// TwinCAT 3 PLC project tc_project_app
// ProgramVersion: 3.1.4026.16
// libraries:
//   Tc2_EtherCAT, * (Beckhoff Automation GmbH)
//   Tc2_MC2, * (Beckhoff Automation GmbH)
//   Tc2_NC, * (Beckhoff Automation GmbH)
//   Tc2_Standard, * (Beckhoff Automation GmbH)
//   Tc2_SUPS, * (Beckhoff Automation GmbH)
//   Tc2_System, * (Beckhoff Automation GmbH)
//   Tc2_Utilities, * (Beckhoff Automation GmbH)
//   Tc3_MC2_AdvancedHoming, * (Beckhoff Automation GmbH)
//   Tc3_Module, * (Beckhoff Automation GmbH)
//   VisuDialogs, * (System)
//   VisuSymbols,3.5.10.0,System
// project tree:
//   / GlobalTextList.TcGTLO (not stored), PlcTask.TcTTO (not stored), VisualizationManager.TcVMO (not stored)
//   GVLs/ GVL_APP.TcGVL, GVL_AxisNames.TcGVL
//   POUs/Application_Specific/Applications/ Application_Template.TcPOU (not stored), AxisTestProg.TcPOU
//   POUs/ MAIN.TcPOU
//   tc_mca_std_lib/DUTs/Axis_Structures/ ST_AxisConfig.TcDUT (not stored), ST_AxisControl.TcDUT (not stored), ST_AxisDescription.TcDUT (not stored), ST_AxisError.TcDUT (not stored), ST_AxisHomingConfig.TcDUT (not stored), ST_AxisInputs.TcDUT (not stored), ST_AxisPersistent.TcDUT (not stored), ST_AxisSPG.TcDUT (not stored), ST_AxisStatus.TcDUT (not stored), ST_AxisStruct.TcDUT (not stored)
//   tc_mca_std_lib/DUTs/ E_AxisParameters.TcTLEO (not stored), E_HomingRoutines.TcTLEO (not stored), E_AxisParameters.TcTLEO (not stored), E_RestorePosition.TcDUT (not stored), I_Axis.TcIO (not stored), E_SlitPairStatesV2.TcDUT (not stored), E_SlitPairStates.TcDUT (not stored), E_MotionFunctions.TcDUT (not stored), ST_McStatus.TcDUT (not stored)
//   tc_mca_std_lib/DUTs/Pneumatics/ E_PneumaticAxisErrors.TcDUT (not stored), E_PneumaticMode.TcDUT (not stored), ST_PneumaticAxisControl.TcDUT (not stored), ST_PneumaticAxisConfig.TcDUT (not stored), ST_PneumaticAxisInputs.TcDUT (not stored), ST_PneumaticAxisOutputs.TcDUT (not stored), ST_PneumaticAxisStatus.TcDUT (not stored), ST_PneumaticAxisStruct.TcDUT (not stored)
//   tc_mca_std_lib/GVLs/ GVL.TcGVL (not stored), GVL_UnitStrings.TcGVL (not stored)
//   tc_mca_std_lib/POUs/Motion/ FB_Axis.TcPOU, FB_SlitPair.TcPOU (not stored), FB_SlitPairV2.TcPOU (not stored), FB_SlitPairV3.TcPOU (not stored)
//   tc_mca_std_lib/POUs/Motion/Homing/ FB_Homing.TcPOU (not stored)
//   tc_mca_std_lib/POUs/Pneumatics/ FB_PneumaticAxis.TcPOU (not stored)
//   tc_mca_std_lib/Unused ESS Work/ E_AxisEngUnit.TcDUT (not stored), E_MonitoringLedFunction.TcDUT (not stored), FB_AxisTemperature.TcPOU (not stored), FB_ESSMonitoring.TcPOU (not stored), ST_MonitoringAlarm.TcDUT (not stored)
//   tc_mca_std_lib/VISUs/ MainVisu.TcVIS, ParameterTextList.TcTLO (not stored), PneumaticsVisu.TcVIS
// real-time tasks:
//   TASK PlcTask: cycle T#2ms, priority 10, ADS port 351
// motion (NC):
//   TASK NC-Task 1 SAF: cycle T#2ms, priority 4, ADS port 501
//   TASK NC-Task 1 SVB: cycle T#10ms, priority 8, ADS port 511
//   AXIS Axis 2 (id 2)
//     Dynamic: Acceleration=600, Deceleration=600
//     Velo: SlowManual=1, FastManual=3, Maximum=6
//     TargetPosControl: Range=0.005, Time=0.2
//     OtherSettings: AllowMotionCmdToSlave=true
//     encoder EncType=19
//       EncPara: ScaleFactorNumerator=5e-05, Offset=-351.3178, MaxCount=#xffffffff, ReferenceSystem=1
//         Inc: RefSoftSyncMask=#xffffffff
//     drive DrvType=24
//       Analog: VeloReferenz=6.25, VeloScale=0.95, TorqueSetpointScale=10, ScaleFactorActTorque=0.1
//       TimeComp: TaskDelayCycles=1
//     controller CtrType=1
//       CtrPara: PriorControlFactor=1
//         PosDiffControl: Range=1.5
//         PID: PosKp=4
//         Observer: BandWidth=20
// I/O:
//   DEVICE Device 1 (EtherCAT), AmsNetId 5.79.68.132.2.1
//     Term 1 (EK1200) [EK1200-5000 EtherCAT Power supply (2A E-Bus)]
//       Term 2 (EL1088) [EL1088 8Ch. Dig. Input 24V, 3ms, negative]
//       Term 3 (EL1808)
//       Term 4 (EL2819) [EL2819 16Ch. Dig. Output 24V, 0,5A, Diagnostic]
//       Term 5 (EK1110) [EK1110 EtherCAT extension]
//     Term 6 (EK1100) [EK1100 EtherCAT Coupler (2A E-Bus)]
//       Term 7 (EL3214) [EL3214 4Ch. Ana. Input PT100 (RTD)]
//       Term 8 (EL7047) [EL7047 1Ch. Stepper motor output stage (50V, 5A)]
//       Term 9 (EL7047) [EL7047 1Ch. Stepper motor output stage (50V, 5A)]
//       Term 10 (EL2008) [EL2008 8Ch. Dig. Output 24V, 0.5A]
//       Term 11 (EL7041-0052) [EL7041-0052 1Ch. Stepper motor output stage (50V, 5A)]
//       Term 12 (EL7041-1000) [EL7041-1000 1Ch. Stepper motor output stage (50V, 5A, standard)]
//       Term 13 (EL5042) [EL5042 2Ch. BiSS-C Encoder]
//       Term 28 (EL2008) [EL2008 8Ch. Dig. Output 24V, 0.5A]
//       Term 29 (EL1008) [EL1008 8Ch. Dig. Input 24V, 3ms]
//       Term 14 (EL9011) [EL9011 End Terminal]
// variable links:
//   (this object) <-> Device 1 (EtherCAT)/Term 6 (EK1100)/Term 13 (EL5042)
//     Enc/Inputs/In/nDataIn1 <-> FB Inputs Channel 1 compact/Position
//     Enc/Inputs/In/nState1 @bit 1 <-> FB Inputs Channel 1 compact/Status/Error
//     Enc/Inputs/In/nState1 @bit 2 <-> FB Inputs Channel 1 compact/Status/Ready
//     Enc/Inputs/In/nState1 <-> FB Inputs Channel 1 compact/Status/Warning
//     Enc/Inputs/In/nState2 @bit 4 <-> FB Inputs Channel 1 compact/Status/Diag
//     Enc/Inputs/In/nState2 @bit 6 <-> FB Inputs Channel 1 compact/Status/Input cycle counter
//     Enc/Inputs/In/nState2 @bit 5 <-> FB Inputs Channel 1 compact/Status/TxPDO State
//     Enc/Inputs/In/nState4 @bit 1 <-> WcState/InputToggle
//     Enc/Inputs/In/nState4 <-> WcState/WcState
//   (this object) <-> Device 1 (EtherCAT)/Term 6 (EK1100)/Term 9 (EL7047)
//     Drive/Inputs/In/nState1 @bit 3 <-> STM Status/Status/Error
//     Drive/Inputs/In/nState1 @bit 7 <-> STM Status/Status/Motor stall
//     Drive/Inputs/In/nState1 @bit 5 <-> STM Status/Status/Moving negative
//     Drive/Inputs/In/nState1 @bit 4 <-> STM Status/Status/Moving positive
//     Drive/Inputs/In/nState1 @bit 1 <-> STM Status/Status/Ready
//     Drive/Inputs/In/nState1 <-> STM Status/Status/Ready to enable
//     Drive/Inputs/In/nState1 @bit 6 <-> STM Status/Status/Torque reduced
//     Drive/Inputs/In/nState1 @bit 2 <-> STM Status/Status/Warning
//     Drive/Inputs/In/nState2 @bit 3 <-> STM Status/Status/Digital input 1
//     Drive/Inputs/In/nState2 @bit 4 <-> STM Status/Status/Digital input 2
//     Drive/Inputs/In/nState2 @bit 5 <-> STM Status/Status/Sync error
//     Drive/Inputs/In/nState2 @bit 7 <-> STM Status/Status/TxPDO Toggle
//     Drive/Inputs/In/nState4 @bit 1 <-> WcState/InputToggle
//     Drive/Inputs/In/nState4 <-> WcState/WcState
//     Drive/Outputs/Out/nCtrl1 <-> STM Control/Control/Enable
//     Drive/Outputs/Out/nCtrl1 @bit 2 <-> STM Control/Control/Reduce torque
//     Drive/Outputs/Out/nCtrl1 @bit 1 <-> STM Control/Control/Reset
//     Drive/Outputs/Out/nCtrl2 @bit 3 <-> STM Control/Control/Digital output 1
//     Drive/Outputs/Out/nDataOut2[0] <-> STM Velocity/Velocity
//   tc_project_app Instance <-> Device 1 (EtherCAT)/Term 6 (EK1100)/Term 28 (EL2008)
//     PlcTask Outputs/AxisTestProg.limitsPower <-> Channel 1/Output
//   tc_project_app Instance <-> Device 1 (EtherCAT)/Term 6 (EK1100)/Term 29 (EL1008)
//     PlcTask Inputs/GVL.astAxes[1].stInputs.bLimitBwd <-> Channel 2/Input
//     PlcTask Inputs/GVL.astAxes[1].stInputs.bLimitFwd <-> Channel 1/Input
//   tc_project_app Instance <-> NC-Task 1 SAF/Axes/Axis 2
//     PlcTask Inputs/GVL.astAxes[1].Axis.NcToPlc <-> Outputs/ToPlc
//     PlcTask Outputs/GVL.astAxes[1].Axis.PlcToNc <-> Inputs/FromPlc

// ---- GVLs/GVL_APP.TcGVL
{attribute 'qualified_only'}
VAR_GLOBAL
END_VAR

VAR_GLOBAL CONSTANT
    nAXIS_NUM: UINT := 8;
    nPNEUMATIC_AXIS_NUM: UINT := 0;
END_VAR

// ---- GVLs/GVL_AxisNames.TcGVL
VAR_GLOBAL
	MEASUREMENT_ANGLE : UINT := 1;
	HEIGHT_VIRTUAL : UINT:= 2;
	HEIGHT : UINT := 3;
	HORIZONTAL : UINT := 4;
	HORIZONTAL_VIRTUAL : UINT := 5;
	ROTATION_VIRTUAL : UINT := 6;
	ROTATION_LINEAR_REAL : UINT := 7;
	ROTATION_LINEAR_VIRTUAL_ENCODER : UINT := 8; //Encoder only axis to get speed information from
END_VAR

// ---- POUs/Application_Specific/Applications/AxisTestProg.TcPOU
PROGRAM AxisTestProg
VAR
    limitsPower AT %Q*: BOOL :=TRUE;
END_VAR

astAxes[1].stControl.bEnable:= TRUE;

END_PROGRAM

// ---- POUs/MAIN.TcPOU
PROGRAM MAIN
VAR
    sVersion: STRING := '1.0.0';
    aIAxes: ARRAY [1..GVL_APP.nAXIS_NUM] OF I_Axis;
    afbAxes: ARRAY [1..GVL_APP.nAXIS_NUM] OF FB_Axis;
    afbPneumaticAxes: ARRAY [1..GVL_APP.nPNEUMATIC_AXIS_NUM] OF FB_PneumaticAxis;
    hmiAxisSelection: INT := 1; //Not possible to use local hmi variables for array indexes
    hmiPneumaticAxisSelection: INT := 1;
//Startup, Shutdown and UPS
    fbUPS: FB_S_UPS_CX51x0;
    eUpsMode: E_S_UPS_Mode := eSUPS_WrPersistData_Shutdown;
    eStartUp: (eColdStart, eReadAxisFeedbackType, eCheckReadDone, eExecuteRestore, eCheckRestore, eFinishRestore);
    bPositionRestoreDone: BOOL := FALSE;
    bRestoreExecute: BOOL := FALSE;
	restoreCounter : UINT:=0;
	restoreCounterMax: UINT:=10;
    bExecuteReadEncRefSys: BOOL := FALSE;
    nRetry: INT;
    iAxes: UINT; //index for for loops in Position recovery actions
    afbReadEncRefSys: ARRAY [1..GVL_APP.nAXIS_NUM] OF MC_ReadParameter;
    afbSetPosition: ARRAY [1..GVL_APP.nAXIS_NUM] OF MC_SetPosition;
    afbReadPositionBias: ARRAY [1..GVL_APP.nAXIS_NUM] OF MC_ReadParameter;
    afbWritePositionBias: ARRAY [1..GVL_APP.nAXIS_NUM] OF MC_WriteParameter;
    fbGetDeviceIdentification: FB_GetDeviceIdentificationEx;
		
    tempAXOutput AT%Q* : BOOL:= TRUE;
	
	
END_VAR

VAR PERSISTENT
    bRestoreOnStartup: BOOL := TRUE;
END_VAR

//POSITION_RECOVERY();
RESTORE_POSITIONS();


IF bPositionRestoreDone THEN
	STORE_PERSISTENT();
END_IF


PROG();
AXES();

ACTION AXES:
//First cycle, assign FB_axis to interface array
IF _TaskInfo[fbGetCurTaskIndex.index].FirstCycle THEN
    FOR GVL.iAxis := 1 TO GVL_APP.nAXIS_NUM DO
        afbAxes[GVL.iAxis].stAxis REF= astAxes[GVL.iAxis];
        aIAxes[GVL.iAxis] := afbAxes[GVL.iAxis];
    END_FOR
    //Custom axis types defined and linked to aiAxes here
      //FB_CustomAxis extends FB_axis
        //fbCustomAxis.stAxis REF= astAxes[x];
        //aIAxes[x] := fbCustomAxis;
END_IF

//Execute FB_Axis logic
FOR GVL.iAxis := 1 TO GVL_APP.nAXIS_NUM DO
    aIAxes[GVL.iAxis].Run();
END_FOR

//Execute Pneumatic Axis logic
FOR GVL.iPneumaticAxis := 1 TO GVL_APP.nPNEUMATIC_AXIS_NUM DO
    afbPneumaticAxes[GVL.iPneumaticAxis](stPneumaticAxisStruct := GVL.astPneumaticAxes[GVL.iPneumaticAxis]);
END_FOR
END_ACTION

ACTION CHECK_UPS:
fbUPS(eUpsMode := eUpsMode);

FOR iAxes := 1 TO GVL_APP.nAXIS_NUM DO
    //Read encoder position BIAS
    IF astAxes[iAxes].stStatus.bAxisInitialized THEN
        afbReadPositionBias[iAxes](Axis := GVL.astAxes[iAxes].Axis,
                        Enable := TRUE,
                        ReadMode:= READMODE_CYCLIC,
                        ParameterNumber := E_AxisParameters.AxisEncoderOffset);
    END_IF
END_FOR

IF eGlobalSUpsState = eSUPS_PowerFailure THEN
    //first cycle of powerfailure
    //execute code that should only be done once with each powerfailure, i.e. increase powerfailure counter
    bRestoreOnStartup := TRUE;
    STORE_PERSISTENT();
    RETURN;
ELSIF eGlobalSUpsState <> eSUPS_PowerOK THEN
    //next cycles of powerfailure
    //skip regular code execution for the remaining cycles of the powerfailure/writing of persistent data/quick shutdown...
    RETURN;
END_IF
END_ACTION

ACTION POSITION_RECOVERY:
fbGetDeviceIdentification(bExecute := TRUE);
IF (fbGetDeviceIdentification.stDevIdent.strHardwareSerialNo <> '') THEN
    CHECK_UPS();
    RESTORE_POSITIONS();
END_IF
END_ACTION

ACTION PROG:
//Get task index for Axes parameters initialization.
GVL.fbGetCurTaskIndex();

//Call the programs that are defined in the "Application Specific" folder.
//Create as many programs in that folder as axes and applications you have or need

//Axes initial parameters and program
//Axis_Template();
//Pneumatics_Template();

//Application program calls
//Application_Template();
AxisTestProg();
END_ACTION

ACTION RESTORE_POSITIONS:
//This ACT will restore the position of an incremental axis on startup with the act position it read before losing power.
//It checks the type of axis, 0=incremental, and that the axis was stationary at shut down.
//Because 0 equates to incremental we also need to check that the data is valid, otherwise by default it would restore all axes.
//By default an axis will not restore the position unless it is set to opt-in, i.e. GVL.aAxes[iAxes].stConfig.eRestorePosition is non-zero.
//This needs to be initialised somewhere in TwinCAT code otherwise it will not be available at start up.
//A restore will only be performed on a loss of power, this code shouldn't make any changes on a reset cold, a rest origin or a download.
//There is a enum to allow for different types of restore modes, currently only one is implemented.
//0 'DontRestore'
//1 'RestoreWithoutHome' -restores the position using a set position fb and does not set the home bit in the axis struct.
//Note from Beckhoff: "A maximum of 1 MB persistent data can be reliably saved over the entire service life."
//Encoder Reference system types: https://infosys.beckhoff.com/english.php?content=../content/1033/tf50x0_tc3_nc_ptp/3439907723.html&id=
//INCREMENTAL=0;
//ABSOLUTE=1;
//ABSOLUTE (modulo)=2;
//ABSOLUTE MULTITURN RANGE (with single overflow)=3;
//INCREMENTAL (singleturn absolute)=4;
//ABSOLUTE SINGLETURN RANGE (with single overflow)=5;

IF NOT bPositionRestoreDone THEN
	bRestoreExecute := TRUE;
END_IF

//IF bRestoreOnStartup AND eGlobalSUpsState = eSUPS_PowerOK THEN
//    bRestoreOnStartup := FALSE;
//    bRestoreExecute := TRUE;
//END_IF

//Upon startup bPositionRestoreDone will be set to FALSE, after successfully completing the following code it will be set TRUE
//and should stay TRUE for the rest of the time the PLC is operational, thus this routine should only be completed once.
IF bRestoreExecute AND NOT bPositionRestoreDone THEN
    //Cycle through function blocks that read the encoder reference system i.e. whether axis is incremental or absolute
    FOR iAxes := 1 TO GVL_APP.nAXIS_NUM DO
         afbReadEncRefSys[iAxes](
            Axis := GVL.astAxes[iAxes].Axis,
            ParameterNumber := MC_AxisParameter.AxisEncoderReferenceSystem,
            ReadMode := E_READMODE.READMODE_ONCE);
    END_FOR

    //Cycle through set position and MC_WritePArameter function blocks for each axis
    FOR iAxes := 1 TO GVL_APP.nAXIS_NUM DO
        afbSetPosition[iAxes](
            Axis := GVL.astAxes[iAxes].Axis,
            Position := astAxesPersistent[iAxes].fPositionAtShutdown);

        afbWritePositionBias[iAxes](
            Axis:= GVL.astAxes[iAxes].Axis,
            ParameterNumber:= E_AxisParameters.AxisEncoderOffset,
            Value:= astAxesPersistent[iAxes].fEncoderBiasAtShutdown);
    END_FOR

    CASE eStartUp OF
        eColdStart:
            //First cycle of the PLC, do nothing just give one cycle for variables to initialise
            IF NOT bPositionRestoreDone THEN
                eStartUp := eReadAxisFeedbackType;
                nRetry := 0;
            END_IF

        eReadAxisFeedbackType:
            //Exectute the function blocks to read the encoder reference system (0=inc OR 1=ABS)
            FOR iAxes := 1 TO GVL_APP.nAXIS_NUM DO
                afbReadEncRefSys[iAxes].Enable := TRUE;
                eStartUp := eCheckReadDone;
            END_FOR

        eCheckReadDone:
            //Check the encoder reference system has been read for all axis -> if busy then continue with PLC cycle and check again next time.
            //If afbReadEncRefSys not started then go back a step.
            //If any axes result in an error the code will get stuck here, this happens if GVL_APP.nAXIS_NUM is not set correctly
            FOR iAxes := 1 TO GVL_APP.nAXIS_NUM DO
                IF NOT afbReadEncRefSys[iAxes].Valid THEN
                    IF afbReadEncRefSys[iAxes].Busy THEN
                        //Exit MAIN.STARTUP Action and wait till next cycle, needs to cycle through whole program in order for data to update
                        RETURN;
                    ELSE
                        //Sometimes the code gets here and the afbReadEncRefSys[iAxes] misses the rising edge. If  the code gets here it means
                        //valid=FALSE and .busy=FALSE which indicateds the FB probably hasn't started and thus needs to see a rising edge.
                        //Set execute to low, Exit MAIN.STARTUP and go back a step in the CASE statement.
                        afbReadEncRefSys[iAxes].Enable := FALSE;
                        eStartUp := eReadAxisFeedbackType;
                        nRetry := nRetry + 1; //counter used for troubleshooting to see how many cycles it takes before afbReadEncRefSys function blocks are read correctly
                        RETURN;
                    END_IF
                END_IF
            END_FOR
            //If the code gets here all axes have .valid=TRUE for all axes
            eStartUp := eExecuteRestore;

        eExecuteRestore:
            //Execute position and encoder BIAS restore by setting Execute = TRUE
           FOR iAxes := 1 TO GVL_APP.nAXIS_NUM DO
                IF GVL.astAxes[iAxes].stConfig.eRestorePosition = E_RestorePosition.eRestoreWithoutHome THEN
                    //Restore position value for incremental encoders
                    IF afbReadEncRefSys[iAxes].Value = 1 OR
                    afbReadEncRefSys[iAxes].Value = 3 OR
                    afbReadEncRefSys[iAxes].Value = 5 THEN
                       afbWritePositionBias[iAxes].Execute := TRUE;
					ELSIF NOT astAxesPersistent[iAxes].bMovingAtShutdown THEN
                       afbSetPosition[iAxes].Execute := TRUE;
                    //Restore encoder position BIAS for absolute encoders
                    
                    END_IF
                ELSE
                    RETURN;
                END_IF
            END_FOR
			restoreCounter:= restoreCounter+1;
            eStartUp := eCheckRestore;


        eCheckRestore:
            //Check the set position and write enocder BIAS fbs are finished
            //Nothing actually happens if the restore is not done, the code just returns from here each cycle and the
            //bPositionRestoreDone will never get set to TRUE and will take up cycle time
			IF restoreCounter>restoreCounterMax THEN
				eStartUp:= eFinishRestore;
				RETURN;
			END_IF
            eStartUp:= eFinishRestore;
			FOR iAxes := 1 TO GVL_APP.nAXIS_NUM DO
				
                IF GVL.astAxes[iAxes].stConfig.eRestorePosition = E_RestorePosition.eRestoreWithoutHome THEN
                    IF afbReadEncRefSys[iAxes].Value = 1 OR
                     afbReadEncRefSys[iAxes].Value = 3 OR
                     afbReadEncRefSys[iAxes].Value = 5 THEN
                        IF NOT afbWritePositionBias[iAxes].Done THEN
                            afbWritePositionBias[iAxes].Execute := FALSE;
                            eStartUp := eExecuteRestore;
                            RETURN;
                        END_IF
					ELSIF NOT astAxesPersistent[iAxes].bMovingAtShutdown THEN 
                        IF NOT afbSetPosition[iAxes].Done THEN
                            afbSetPosition[iAxes].Execute := FALSE;
                            eStartUp := eExecuteRestore;
                            RETURN;
                        END_IF
                     
                    END_IF
                END_IF
            END_FOR
            

        eFinishRestore:
            //Remove execute = TRUE for afbRestorePosition and fbWritePositionBias
            FOR iAxes := 1 TO GVL_APP.nAXIS_NUM DO
                afbSetPosition[iAxes].Execute := FALSE;
                afbWritePositionBias[iAxes].Execute := FALSE;
                bPositionRestoreDone := TRUE;
                bRestoreExecute := FALSE;
            END_FOR
    END_CASE
END_IF
END_ACTION

ACTION STORE_PERSISTENT:
FOR iAxes := 1 TO GVL_APP.nAXIS_NUM DO
    //Store Position beofre shutdown
    astAxesPersistent[iAxes].fPositionAtShutdown := GVL.astAxes[iAxes].Axis.NcToPlc.ActPos;

    //Store encoder position BIAS at shutdown
    astAxesPersistent[iAxes].fEncoderBiasAtShutdown := afbReadPositionBias[iAxes].Value;

    //Store value of moving at shutdown
    IF GVL.astAxes[iAxes].Axis.Status.StandStill OR GVL.astAxes[iAxes].Axis.Status.Disabled THEN
        astAxesPersistent[iAxes].bMovingAtShutdown := FALSE;
    ELSE
        astAxesPersistent[iAxes].bMovingAtShutdown := TRUE;
    END_IF
END_FOR
END_ACTION

END_PROGRAM

// ---- tc_mca_std_lib/POUs/Motion/FB_Axis.TcPOU
//Function block to run a virtual drive with Nc
FUNCTION_BLOCK FB_Axis IMPLEMENTS I_axis
VAR
    _stAxis: REFERENCE TO ST_AxisStruct; // Local property pointer for axis structure
    astMcStatus: ARRAY[1..nMCSTATUS_ARRAY_SIZE] OF POINTER TO ST_McStatus; //Array of all MC status signals defined in FB_init

    fbPower: MC_Power;
    stMcStatusPower: ST_McStatus;

    fbStop: MC_Stop;
    stMcStatusStop: ST_McStatus;

    fbHalt: MC_Halt;
    stMcStatusHalt: ST_McStatus;

    fbReset: MC_Reset;
    stMcStatusReset: ST_McStatus;

    fbMoveAbsolute: MC_MoveAbsolute;
    fbMoveAbsolute2: MC_MoveAbsolute;
    stMcStatusMoveAbsolute: ST_McStatus;

    fbMoveRelative: MC_MoveRelative;
    stMcStatusMoveRelative: ST_McStatus;

    fbMoveVelocity: MC_MoveVelocity;
    stMcStatusMoveVelocity: ST_McStatus;

    fbMoveModulo: MC_MoveModulo;
    fbMoveModulo2: MC_MoveModulo;
    stMcStatusMoveModulo: ST_McStatus;
	
	fbEnableSPG : MC_ExtSetPointGenEnable;
	stMcStatusEnableSPG : ST_McStatus;
	fbDisableSPG : MC_ExtSetPointGenDisable;
	stMcStatusDisableSPG : ST_McStatus;
	

    fbHome: FB_Homing;
    stMcStatusHome: ST_McStatus;

    fbReadParameter: MC_ReadParameter;
    stMcStatusReadParameter: ST_McStatus;

    fbWriteParameter: MC_WriteParameter;
    stMcStatusWriteParameter: ST_McStatus;
	
	fbSetPosition: MC_SetPosition;
	stMcStatusSetPosition: ST_McStatus;

    //Variables for holding limits during homing
    bWaitForStopAfterLimitHit: BOOL := FALSE;
    fbRemovePowerTimer: TOF;

    //Dedicated NC parameter read FBs
    fbReadAxisVeloManSlow: MC_ReadParameter;
    fbReadAxisVeloManFast: MC_ReadParameter;
    fbReadHomingVelToCam: MC_ReadParameter;
    fbReadHomingVelFromCam: MC_ReadParameter;
    fbReadAxisVeloMax: MC_ReadParameter;
    fbReadAxisMaxAcc: MC_ReadParameter;
    fbReadAxisMaxDec: MC_ReadParameter;
    fbReadAxisAcc: MC_ReadParameter;
    fbReadAxisDec: MC_ReadParameter;
    fbReadEnMinSoftPosLimit: MC_ReadParameter;
    fbReadEnMaxSoftPosLimit: MC_ReadParameter;
    fbReadMinSoftPosLimit: MC_ReadParameter;
    fbReadMaxSoftPosLimit: MC_ReadParameter;
    fbReadEnPositionLagMonitoring: MC_ReadParameter;
    fbReadAxisMaxPosLagValue: MC_ReadParameter;
    fbReadEnTargetPositionMonitoring: MC_ReadParameter;
    fbReadTargetPositionWindow: MC_ReadParameter;

    //Edge detection triggers for statuses
    fbDoneRTrig: R_TRIG;
    fbErrorRTrig: R_TRIG;
    fbCommandAbortedRTrig: R_TRIG;
    fbInVelocityRTrig: R_TRIG;
    fbInVelocityFTrig: F_TRIG;
    fbExecuteRTrig: R_TRIG;
    fbStopFinishedRiseEdge: R_TRIG;
    fbHaltFinishedRiseEdge: R_TRIG;
    fbResetFinishedRiseEdge: R_TRIG;
    fbAbsMovDyn1RiseEdge: R_TRIG;
    fbAbsMovDyn2RiseEdge: R_TRIG;
    fbModMovDyn1RiseEdge: R_TRIG;
    fbModMovDyn2RiseEdge: R_TRIG;
	
	fbMoveInProgressFTrig : F_TRIG;
	fbMoveInProgressEndTimer : TON;
	fbNewMoveRTrig : R_TRIG;
	bStartOfMove : BOOL;
	bEndOfMove : BOOL;
	
	bSpgEnableReq : BOOL;
	bSpgDisableReq : BOOL;
	spgDisableCommand : BOOL;

END_VAR
VAR CONSTANT
    nRATIO_DENOMINATOR_DEFAULT: UINT := 1;
    nNO_GEARING: UINT := 0;
    nMCSTATUS_ARRAY_SIZE: UINT := 12;
    nMULTI_MASTER_MAX_AXES: UINT := 4;
END_VAR

METHOD EndOfCycle : BOOL

_stAxis.stControl.bExecute := FALSE;
END_METHOD

METHOD FB_init : BOOL
VAR_INPUT
    bInitRetains: BOOL; // if TRUE, the retain variables are initialized (warm start / cold start)
    bInCopyCode: BOOL; // if TRUE, the instance afterwards gets moved into the copy code (online change)
END_VAR

//Copy address locations for statuses to an array to allow for easier checking of statuses
astMcStatus[1] := ADR(stMcStatusPower);
astMcStatus[2] := ADR(stMcStatusStop);
astMcStatus[3] := ADR(stMcStatusHalt);
astMcStatus[4] := ADR(stMcStatusReset);
astMcStatus[5] := ADR(stMcStatusMoveAbsolute);
astMcStatus[6] := ADR(stMcStatusMoveRelative);
astMcStatus[7] := ADR(stMcStatusMoveVelocity);
astMcStatus[8] := ADR(stMcStatusMoveModulo);
astMcStatus[9] := ADR(stMcStatusHome);
astMcStatus[10] := ADR(stMcStatusSetPosition);
astMcStatus[11] := ADR(stMcStatusReadParameter);
astMcStatus[12] := ADR(stMcStatusWriteParameter);
END_METHOD

METHOD mControl_AutoEnableDisable : BOOL
VAR_INPUT
END_VAR
//Has a move been requested?
IF _stAxis.stControl.eCommand = E_MotionFunctions.eMoveAbsolute OR 
	_stAxis.stControl.eCommand = E_MotionFunctions.eMoveModulo OR
	_stAxis.stControl.eCommand = E_MotionFunctions.eMoveRelative OR
	_stAxis.stControl.eCommand = E_MotionFunctions.eMoveVelocity OR
	_stAxis.stControl.eCommand = E_MotionFunctions.eHome THEN
	IF _stAxis.stControl.bExecute AND _stAxis.stStatus.bMoveRequested = FALSE THEN
		//new logic here to stop commands queuing with axes disabled if not meant to autoenable/disable
 		IF _stAxis.stStatus.bEnabled = FALSE AND _stAxis.stControl.bAutoEnableDisable = FALSE THEN
			_stAxis.stStatus.bMoveRequested := FALSE;
		ELSE
			_stAxis.stStatus.bMoveRequested := TRUE;
		END_IF
		//_stAxis.stStatus.bMoveRequested := TRUE;
	END_IF	
END_IF

IF _stAxis.stControl.bOverrideReadyToMove THEN
	_stAxis.stStatus.bReadyToMove := _stAxis.stControl.bExtReadyToMove;
ELSE
	_stAxis.stStatus.bReadyToMove := _stAxis.stStatus.bEnabled;
END_IF

IF fbMoveInProgressFTrig.Q THEN
	//start end move timer
	bEndOfMove:= TRUE;
	_stAxis.stControl.bExtReadyToMove:= FALSE;
END_IF
IF bStartOfMove THEN
	bEndOfMove:= FALSE;
	bStartOfMove:= FALSE;
END_IF

fbMoveInProgressEndTimer(IN:= bEndOfMove,PT:= _stAxis.stControl.tMoveFinishedDelay);

//If we want autoenabledisable
IF _stAxis.stControl.bAutoEnableDisable THEN
	//and a move has been requested and we are not enabled
	IF _stAxis.stStatus.bMoveRequested AND _stAxis.stStatus.bEnabled = FALSE THEN
		_stAxis.stControl.bEnable:= TRUE;
	END_IF
	IF _stAxis.stStatus.bMoveRequested = FALSE AND fbMoveInProgressEndTimer.Q THEN
	_stAxis.stControl.bEnable:= FALSE;
	bEndOfMove := FALSE;
	END_IF
END_IF

IF _stAxis.Axis.Status.Moving THEN
	_stAxis.stStatus.bMoveInProgress := TRUE;
END_IF

IF _stAxis.Axis.Status.NotMoving THEN
	_stAxis.stStatus.bMoveInProgress := FALSE;
END_IF

fbNewMoveRTrig(CLK:= _stAxis.stStatus.bMoveInProgress);
IF fbNewMoveRTrig.Q THEN
	bStartOfMove:= TRUE;
END_IF
fbMoveInProgressFTrig(CLK:= _stAxis.stStatus.bMoveInProgress OR spgDisableCommand);
//No move requested and no move in progress
END_METHOD

METHOD mControl_DisableSPG : BOOL
VAR_INPUT
END_VAR
IF _stAxis.stSpg.DisableSPG THEN
	//fbEnableSPG.Execute := TRUE;
	bSpgDisableReq := TRUE;
END_IF

IF _stAxis.stStatus.bEnabled = FALSE AND bSpgDisableReq THEN
	_stAxis.stStatus.messageString:= 'Axis is disabled';
	bSpgDisableReq:= FALSE;
END_IF

IF _stAxis.stStatus.SPGEnabled = FALSE AND bSpgDisableReq THEN
	stAxis.stStatus.messageString:= 'Axis is not in ExtSPG mode';
	bSpgDisableReq:= FALSE;
END_IF





fbDisableSPG.Execute:= bSpgDisableReq;
fbDisableSPG(Axis:= _stAxis.Axis);
IF _stAxis.stControl.bAutoEnableDisable THEN
	spgDisableCommand := fbDisableSPG.Done;
END_IF

_stAxis.stSpg.DisableSPG:= FALSE;
fbDisableSPG.Execute := FALSE;
END_METHOD

METHOD mControl_EnableSPG : BOOL
VAR_INPUT
END_VAR
IF _stAxis.stSpg.EnableSPG THEN
	//fbEnableSPG.Execute := TRUE;
	bSpgEnableReq := TRUE;
END_IF

IF _stAxis.stControl.bAutoEnableDisable = FALSE AND _stAxis.stStatus.bEnabled = FALSE AND bSpgEnableReq THEN
	_stAxis.stStatus.messageString:= 'Axis must be enabled before enabling ExtSPG';
	bSpgEnableReq:= FALSE;
END_IF

IF _stAxis.stControl.bAutoEnableDisable  AND _stAxis.stStatus.bEnabled = FALSE AND bSpgEnableReq = TRUE THEN
	_stAxis.stControl.bEnable:= TRUE;
END_IF


IF _stAxis.stStatus.bEnabled THEN
	fbEnableSPG.Execute := bSpgEnableReq;
	bSpgEnableReq := FALSE;
END_IF

fbEnableSPG(Axis:= _stAxis.Axis);

_stAxis.stSpg.EnableSPG:= FALSE;
fbEnableSPG.Execute := FALSE;
END_METHOD

METHOD mControl_FeedSPG : BOOL
VAR_INPUT
END_VAR

VAR
	DirectionInternal : DINT;
END_VAR
(* 
Direction 1 = Forward
Direction -1 = Backward
Direction 0 = Standstill
*)

IF _stAxis.stSpg.OverrideDirection THEN
	DirectionInternal:= _stAxis.stSpg.Direction;
ELSE
	//Direction calculation logic
	IF _stAxis.stSpg.Velocity > ABS(_stAxis.stSpg.VelocityStandstillThreshold) THEN
		DirectionInternal := 1;
	ELSIF _stAxis.stSpg.Velocity < -ABS(_stAxis.stSpg.VelocityStandstillThreshold) THEN
		DirectionInternal := -1;
	ELSE
		DirectionInternal := 0;
	END_IF
END_IF

MC_ExtSetPointGenFeed(
	Axis:= _stAxis.Axis, 
	Position:= _stAxis.stSpg.Position,
	Velocity:= _stAxis.stSpg.Velocity,
	Acceleration:= _stAxis.stSpg.Acceleration,
	Direction:= DirectionInternal);
END_METHOD

METHOD mControl_Home : ST_McStatus
IF _stAxis.stHomingConfig.eHomeSeq = E_HomingRoutines.eNoHoming THEN
    _stAxis.stStatus.bHomed := TRUE;
END_IF

IF _stAxis.stControl.eCommand = E_MotionFunctions.eHome THEN
    fbHome.bExecute := _stAxis.stControl.bExecute;
END_IF


fbHome.eHomeSeq := _stAxis.stHomingConfig.eHomeSeq;
fbHome.fHomePosition := _stAxis.stHomingConfig.fHomePosition;
fbHome.fHomeFinishDistance := _stAxis.stHomingConfig.fHomeFinishDistance;
fbHome(
    Axis := _stAxis.Axis,
    bLimitBwd := _stAxis.stInputs.bLimitBwd,
    bLimitFwd := _stAxis.stInputs.bLimitFwd,
    bHomeSensor := _stAxis.stInputs.bHomeSensor,
    stConfig := _stAxis.stConfig);
fbHome.bExecute := FALSE;

mControl_Home.Busy := fbHome.bBusy;
mControl_Home.CommandAborted := fbHome.bCommandAborted;
mControl_Home.Done := fbHome.bDone;
mControl_Home.Error := fbHome.bError;
mControl_Home.ErrorID := fbHome.nErrorId;

IF fbHome.bError THEN
    _stAxis.stError.nHomeErrorID := fbHome.nErrorID; //Set the error
END_IF
END_METHOD

METHOD mControl_LimitHitTimer : BOOL

//Timer for keeping power on after limit switch hit, needed for homing routines - if power is lost routines are aborted
fbRemovePowerTimer(IN := _stAxis.stInputs.bLimitFwd AND _stAxis.stInputs.bLimitBwd, PT := T#100MS);

IF stMcStatusHome.Busy AND (fbRemovePowerTimer.Q OR _stAxis.Axis.NcToPlc.AxisState = 5) THEN //5=PHASE_ACCNEG
    bWaitForStopAfterLimitHit := TRUE;
ELSE
    bWaitForStopAfterLimitHit := FALSE;
END_IF
END_METHOD

METHOD mControl_LimitLinking : BOOL

_stAxis.stStatus.bFwEnabled := _stAxis.stInputs.bLimitFwd OR _stAxis.stControl.bOverrideLimits; 
_stAxis.stStatus.bBwEnabled := _stAxis.stInputs.bLimitBwd OR _stAxis.stControl.bOverrideLimits;
_stAxis.stStatus.bInterlockedFwd := _stAxis.stControl.bInterlockFwd;
_stAxis.stStatus.bInterlockedBwd := _stAxis.stControl.bInterlockBwd;
END_METHOD

METHOD mControl_Power : ST_McStatus
fbPower.Enable := _stAxis.stControl.bEnable;

fbPower.Enable_Negative := (_stAxis.stStatus.bBwEnabled OR bWaitForStopAfterLimitHit) AND NOT _stAxis.stStatus.bInterlockedBwd;
fbPower.Enable_Positive := (_stAxis.stStatus.bFwEnabled OR bWaitForStopAfterLimitHit) AND NOT _stAxis.stStatus.bInterlockedFwd;
fbPower.Override := _stAxis.stConfig.fOverride;

fbPower(Axis := _stAxis.Axis);

mControl_Power.Error := fbPower.Error;

IF fbPower.Error THEN
    _stAxis.stError.nPowerErrorID := fbPower.ErrorID; //Set the error
END_IF
END_METHOD

METHOD mControl_Reset : ST_McStatus
VAR
    i: UINT;
END_VAR
fbReset.Execute := _stAxis.stControl.bReset;

fbReset(Axis := _stAxis.Axis);
IF fbReset.Done THEN
    _stAxis.stStatus.bError := FALSE;
	_stAxis.stStatus.bMcError := FALSE;
    FOR i := 1 TO nMCSTATUS_ARRAY_SIZE DO
        //Clear all the errors
        _stAxis.stStatus.nErrorID := 0;
    END_FOR
	_stAxis.stStatus.nMcErrorID := 0;
END_IF

mControl_Reset.Busy := fbReset.Busy;
mControl_Reset.Done := fbReset.Done;
mControl_Reset.Error := fbReset.Error;
mControl_Reset.ErrorID := fbReset.ErrorID;

IF fbReset.Error THEN
    _stAxis.stError.nResetErrorID := fbReset.ErrorID; //Set the error
END_IF

fbResetFinishedRiseEdge(CLK:=fbReset.Done OR fbReset.Error);
IF fbResetFinishedRiseEdge.Q OR fbReset.Done THEN
    _stAxis.stControl.bReset := FALSE;
END_IF
END_METHOD

METHOD mMove_Halt : ST_McStatus
fbHalt.Deceleration := _stAxis.stControl.fDeceleration;
fbHalt.Execute := _stAxis.stControl.bHalt;

fbHalt(Axis := _stAxis.Axis);

mMove_Halt.Busy := fbHalt.Busy;
mMove_Halt.Done := fbHalt.Done;
mMove_Halt.Error := fbHalt.Error;
mMove_Halt.ErrorID := fbHalt.ErrorID;
mMove_Halt.Active := fbHalt.Active;
mMove_Halt.CommandAborted := fbHalt.CommandAborted;

IF fbHalt.Error THEN
    _stAxis.stError.nHaltErrorID := fbHalt.ErrorID; //Set the error
END_IF

//Execution of fbHalt ended
fbHaltFinishedRiseEdge(CLK:=fbHalt.Done OR fbHalt.Error OR fbHalt.CommandAborted);
IF fbHaltFinishedRiseEdge.Q OR fbHalt.Done OR fbHalt.CommandAborted THEN
    _stAxis.stControl.bHalt := FALSE;
END_IF
END_METHOD

METHOD mMove_MoveAbsolute : ST_McStatus
IF _stAxis.stControl.eCommand = E_MotionFunctions.eMoveAbsolute THEN
	IF _stAxis.stStatus.bReadyToMove THEN
		fbMoveAbsolute.Execute := _stAxis.stStatus.bMoveRequested;
		IF _stAxis.stStatus.bMoveRequested THEN
			_stAxis.stStatus.bMoveRequested := FALSE;
		END_IF
    	IF fbMoveAbsolute.Execute AND fbMoveAbsolute.Busy THEN
        	fbMoveAbsolute2.Execute := TRUE;
    	END_IF
	END_IF    
END_IF

// Parameters
fbMoveAbsolute.Position := _stAxis.stControl.fPosition;
fbMoveAbsolute.Velocity := ABS(_stAxis.stControl.fVelocity);
fbMoveAbsolute.Acceleration := _stAxis.stControl.fAcceleration;
fbMoveAbsolute.Deceleration := _stAxis.stControl.fDeceleration;

fbMoveAbsolute2.Position := _stAxis.stControl.fPosition;
fbMoveAbsolute2.Velocity := ABS(_stAxis.stControl.fVelocity);
fbMoveAbsolute2.Acceleration := _stAxis.stControl.fAcceleration;
fbMoveAbsolute2.Deceleration := _stAxis.stControl.fDeceleration;


// Call both move absolute FB
fbMoveAbsolute(Axis := _stAxis.Axis);
fbMoveAbsolute2(Axis := _stAxis.Axis);

//Reset Execute bits
fbMoveAbsolute.Execute := FALSE;
fbMoveAbsolute2.Execute := FALSE;


// STATUS bits
mMove_MoveAbsolute.Active := fbMoveAbsolute.Active OR fbMoveAbsolute2.Active;
mMove_MoveAbsolute.Done := fbMoveAbsolute.Done OR fbMoveAbsolute2.Done;
mMove_MoveAbsolute.Busy := fbMoveAbsolute.Busy OR fbMoveAbsolute2.Busy;
mMove_MoveAbsolute.Error := fbMoveAbsolute.Error OR fbMoveAbsolute2.Error;


// Capture the CommandAborted for first scan if the other absolute move overtakes the current
fbAbsMovDyn1RiseEdge(CLK:= fbMoveAbsolute.Busy AND fbMoveAbsolute2.CommandAborted, Q=>);
fbAbsMovDyn2RiseEdge(CLK:= fbMoveAbsolute2.Busy AND fbMoveAbsolute.CommandAborted, Q=>);
mMove_MoveAbsolute.CommandAborted := (fbMoveAbsolute.CommandAborted AND NOT fbAbsMovDyn2RiseEdge.Q)
                                    OR (fbMoveAbsolute2.CommandAborted AND NOT fbAbsMovDyn1RiseEdge.Q);

// Error IDs
IF fbMoveAbsolute.Error THEN
    _stAxis.stError.nMoveAbsoluteErrorID := fbMoveAbsolute.ErrorID; //Set the error
    mMove_MoveAbsolute.ErrorID := fbMoveAbsolute.ErrorID;
END_IF
IF fbMoveAbsolute2.Error THEN
    _stAxis.stError.nMoveAbsoluteErrorID := fbMoveAbsolute2.ErrorID; //Set the error
    mMove_MoveAbsolute.ErrorID := fbMoveAbsolute2.ErrorID;
END_IF
END_METHOD

METHOD mMove_MoveModulo : ST_McStatus
IF _stAxis.stControl.eCommand = E_MotionFunctions.eMoveModulo THEN
	IF _stAxis.stStatus.bReadyToMove THEN
		fbMoveModulo.Execute := _stAxis.stStatus.bMoveRequested;
		IF _stAxis.stStatus.bMoveRequested THEN
			_stAxis.stStatus.bMoveRequested := FALSE;
		END_IF
    	IF fbMoveModulo.Execute AND fbMoveAbsolute.Busy THEN
        	fbMoveModulo2.Execute := TRUE;
    	END_IF
	END_IF    
END_IF

// Parameters
fbMoveModulo.Position := _stAxis.stControl.fPosition;
fbMoveModulo.Velocity := ABS(_stAxis.stControl.fVelocity);
fbMoveModulo.Acceleration := _stAxis.stControl.fAcceleration;
fbMoveModulo.Deceleration := _stAxis.stControl.fDeceleration;

fbMoveModulo2.Position := _stAxis.stControl.fPosition;
fbMoveModulo2.Velocity := ABS(_stAxis.stControl.fVelocity);
fbMoveModulo2.Acceleration := _stAxis.stControl.fAcceleration;
fbMoveModulo2.Deceleration := _stAxis.stControl.fDeceleration;

// Call both move absolute FB
fbMoveModulo(Axis := _stAxis.Axis);
fbMoveModulo.Execute := FALSE;
fbMoveModulo2(Axis := _stAxis.Axis);
fbMoveModulo2.Execute := FALSE;

// Status bits
mMove_MoveModulo.Active := fbMoveModulo.Active OR fbMoveModulo2.Active;
mMove_MoveModulo.Done := fbMoveModulo.Done OR fbMoveModulo2.Done;
mMove_MoveModulo.Busy := fbMoveModulo.Busy OR fbMoveModulo2.Busy;
mMove_MoveModulo.Error := fbMoveModulo.Error OR fbMoveModulo2.Error;

// Capture the CommandAborted for first scan if the other absolute move overtakes the current
fbModMovDyn1RiseEdge(CLK:= fbMoveModulo.Busy AND fbMoveModulo2.CommandAborted, Q=>);
fbModMovDyn2RiseEdge(CLK:= fbMoveModulo2.Busy AND fbMoveModulo.CommandAborted, Q=>);
mMove_MoveModulo.CommandAborted := (fbMoveModulo.CommandAborted AND NOT fbModMovDyn2RiseEdge.Q)
                                    OR (fbMoveModulo2.CommandAborted AND NOT fbModMovDyn1RiseEdge.Q);

// Error IDs
IF fbMoveModulo.Error THEN
    _stAxis.stError.nMoveModuloErrorID := fbMoveModulo.ErrorID; //Set the error
    mMove_MoveModulo.ErrorID := fbMoveModulo.ErrorID;
END_IF

IF fbMoveModulo2.Error THEN
    _stAxis.stError.nMoveModuloErrorID := fbMoveModulo2.ErrorID; //Set the error
    mMove_MoveModulo.ErrorID := fbMoveModulo2.ErrorID;
END_IF
END_METHOD

METHOD mMove_MoveRelative : ST_McStatus

IF _stAxis.stControl.eCommand = E_MotionFunctions.eMoveRelative THEN
	IF _stAxis.stStatus.bReadyToMove THEN
		fbMoveRelative.Execute := _stAxis.stStatus.bMoveRequested;
		IF _stAxis.stStatus.bMoveRequested THEN
			_stAxis.stStatus.bMoveRequested := FALSE;
		END_IF
	END_IF
END_IF

fbMoveRelative.Distance := _stAxis.stControl.fPosition;
fbMoveRelative.Velocity := ABS(_stAxis.stControl.fVelocity);
fbMoveRelative.Acceleration := _stAxis.stControl.fAcceleration;
fbMoveRelative.Deceleration := _stAxis.stControl.fDeceleration;

fbMoveRelative(Axis := _stAxis.Axis);
fbMoveRelative.Execute := FALSE;

mMove_MoveRelative.Active := fbMoveRelative.Active;
mMove_MoveRelative.Done := fbMoveRelative.Done;
mMove_MoveRelative.Busy := fbMoveRelative.Busy;
mMove_MoveRelative.Error := fbMoveRelative.Error;
mMove_MoveRelative.ErrorID := fbMoveRelative.ErrorID;
mMove_MoveRelative.CommandAborted := fbMoveRelative.CommandAborted;

IF fbMoveRelative.Error THEN
    _stAxis.stError.nMoveRelativeErrorID := fbMoveRelative.ErrorID; //Set the error
END_IF
END_METHOD

METHOD mMove_MoveVelocity : ST_McStatus

IF _stAxis.stControl.eCommand = E_MotionFunctions.eMoveVelocity THEN
	IF _stAxis.stStatus.bReadyToMove THEN
		fbMoveVelocity.Execute := _stAxis.stStatus.bMoveRequested;
		IF _stAxis.stStatus.bMoveRequested THEN
			_stAxis.stStatus.bMoveRequested := FALSE;
		END_IF
	END_IF
END_IF

fbMoveVelocity.Direction := SEL(_stAxis.stControl.fVelocity < 0, MC_Positive_Direction, MC_Negative_Direction);
fbMoveVelocity.Velocity := ABS(_stAxis.stControl.fVelocity);
fbMoveVelocity.Acceleration := _stAxis.stControl.fAcceleration;
fbMoveVelocity.Deceleration := _stAxis.stControl.fDeceleration;

fbMoveVelocity(Axis := _stAxis.Axis);
fbMoveVelocity.Execute:= FALSE;

mMove_MoveVelocity.Active := fbMoveVelocity.Active;
mMove_MoveVelocity.InVelocity := fbMoveVelocity.InVelocity;
mMove_MoveVelocity.Busy := fbMoveVelocity.Busy;
mMove_MoveVelocity.Error := fbMoveVelocity.Error;
mMove_MoveVelocity.ErrorID := fbMoveVelocity.ErrorID;
mMove_MoveVelocity.CommandAborted := fbMoveVelocity.CommandAborted;

IF fbMoveVelocity.Error THEN
    _stAxis.stError.nMoveVelocityErrorID := fbMoveVelocity.ErrorID; //Set the error
END_IF
END_METHOD

METHOD mMove_SetPosition : ST_McStatus
IF _stAxis.stControl.eCommand = E_MotionFunctions.eSetPosition THEN
	fbSetPosition.Execute:= _stAxis.stControl.bExecute;
END_IF

fbSetPosition.Position:= _stAxis.stControl.fPosition;
fbSetPosition.Options.ClearPositionLag:= TRUE;

fbSetPosition(Axis := _stAxis.Axis);
fbSetPosition.Execute:= FALSE;

mMove_SetPosition.Busy := fbSetPosition.Busy;
mMove_SetPosition.Error := fbSetPosition.Error;
mMove_SetPosition.ErrorID := fbSetPosition.ErrorID;
mMove_SetPosition.Done := fbSetPosition.Done;

IF fbSetPosition.Error THEN
    _stAxis.stError.nSetPositionErrorID := fbSetPosition.ErrorID; //Set the error
END_IF
END_METHOD

METHOD mMove_Stop : ST_McStatus
fbStop.Deceleration := _stAxis.stControl.fDeceleration;
fbStop.Execute := _stAxis.stControl.bStop;

fbStop(Axis := _stAxis.Axis);

mMove_Stop.Busy := fbStop.Busy;
mMove_Stop.Done := fbStop.Done;
mMove_Stop.Error := fbStop.Error;
mMove_Stop.ErrorID := fbStop.ErrorID;
mMove_Stop.Active := fbStop.Active;
mMove_Stop.CommandAborted := fbStop.CommandAborted;

IF fbStop.Error THEN
    _stAxis.stError.nStopErrorID := fbStop.ErrorID; //Set the error
END_IF

//Execution of fbStop ended
fbStopFinishedRiseEdge(CLK:=fbStop.Done OR fbStop.Error OR fbStop.CommandAborted);
IF fbStopFinishedRiseEdge.Q THEN
    _stAxis.stControl.bStop := FALSE;
END_IF
END_METHOD

METHOD mParameters_Init : BOOL
IF _stAxis.stControl.bReinitialiseNcParameters THEN
	_stAxis.stStatus.bAxisInitialized := FALSE;
	_stAxis.stControl.bReinitialiseNcParameters := FALSE;
END_IF
IF _stAxis.stConfig.bReadMcParametersValid AND NOT _stAxis.stStatus.bAxisInitialized THEN
    _stAxis.stControl.fAcceleration := _stAxis.stConfig.fDefaultAcc;
    _stAxis.stControl.fDeceleration := _stAxis.stConfig.fDefaultDec;
    _stAxis.stControl.fVelocity := _stAxis.stConfig.fVelocityDefaultFast;
    _stAxis.stControl.fJogVelocity := _stAxis.stConfig.fVelocityDefaultSlow;

    _stAxis.stStatus.bAxisInitialized := TRUE;
END_IF
END_METHOD

METHOD mParameters_ReadNc : BOOL

(*This act reads the MC parameters using an MC_ReadParameter FB FOR each variable
Intended TO be executed once every PLC cycle
Another FB is used TO trasnfer default axis parameters TO the stAxisStruct so
bReadValid is used TO halt that trasnfer UNTIL the parameters have been
read successfully. It may take a couple OF cycles once the PLC starts up.*)

//Slow jogging Velocity
fbReadAxisVeloManSlow(Axis := _stAxis.Axis,
                        Enable := TRUE,
                        ReadMode := READMODE_CYCLIC,
                        ParameterNumber := E_AxisParameters.AxisManualVelocitySlow,
                        Value => _stAxis.stConfig.fVelocityDefaultSlow);
//Fast jogging velocity
fbReadAxisVeloManFast(Axis := _stAxis.Axis,
                        Enable := TRUE,
                        ReadMode := READMODE_CYCLIC,
                        ParameterNumber := E_AxisParameters.AxisManualVelocityFast,
                        Value => _stAxis.stConfig.fVelocityDefaultFast);
//Homing velocity to Cam
fbReadHomingVelToCam(Axis := _stAxis.Axis,
                        Enable := TRUE,
                        ReadMode := READMODE_CYCLIC,
                        ParameterNumber := E_AxisParameters.AxisVelocityToCam,
                        Value => _stAxis.stHomingConfig.fHomingVelToCam);
//Homing velocity from Cam
fbReadHomingVelFromCam(Axis := _stAxis.Axis,
                        Enable := TRUE,
                        ReadMode := READMODE_CYCLIC,
                        ParameterNumber := E_AxisParameters.AxisVelocityFromCam,
                        Value => _stAxis.stHomingConfig.fHomingVelFromCam);
//Max velocity
fbReadAxisVeloMax(Axis := _stAxis.Axis,
                        Enable := TRUE,
                        ReadMode := READMODE_CYCLIC,
                        ParameterNumber := E_AxisParameters.AxisMaxVelocity,
                        Value => _stAxis.stConfig.fVeloMax);
//Max acceleration
fbReadAxisMaxAcc(Axis := _stAxis.Axis,
                        Enable := TRUE,
                        ReadMode := READMODE_CYCLIC,
                        ParameterNumber := E_AxisParameters.AxisMaximumAcceleration,
                        Value => _stAxis.stConfig.fMaxAcc);
//Max deceleration
fbReadAxisMaxDec(Axis := _stAxis.Axis,
                        Enable := TRUE,
                        ReadMode := READMODE_CYCLIC,
                        ParameterNumber := E_AxisParameters.AxisMaximumDeceleration,
                        Value => _stAxis.stConfig.fMaxDec);
//Default acceleration
fbReadAxisAcc(Axis := _stAxis.Axis,
                        Enable := TRUE,
                        ReadMode := READMODE_CYCLIC,
                        ParameterNumber := E_AxisParameters.AxisDefaultAcceleration,
                        Value => _stAxis.stConfig.fDefaultAcc);
//Default deceleration
fbReadAxisDec(Axis := _stAxis.Axis,
                        Enable := TRUE,
                        ReadMode := READMODE_CYCLIC,
                        ParameterNumber := E_AxisParameters.AxisDefaultDeceleration,
                        Value => _stAxis.stConfig.fDefaultDec);

//Soft limits enabled
fbReadEnMinSoftPosLimit(Axis := _stAxis.Axis,
                        Enable := TRUE,
                        ReadMode := READMODE_CYCLIC,
                        ParameterNumber := E_AxisParameters.EnableLimitBackward);
_stAxis.stConfig.bEnMinSoftPosLimit := LREAL_TO_BOOL(fbReadEnMinSoftPosLimit.Value);

fbReadEnMaxSoftPosLimit(Axis := _stAxis.Axis,
                        Enable := TRUE,
                        ReadMode := READMODE_CYCLIC,
                        ParameterNumber := E_AxisParameters.EnableLimitForward);
_stAxis.stConfig.bEnMaxSoftPosLimit := LREAL_TO_BOOL(fbReadEnMaxSoftPosLimit.Value);

//Soft limit values
fbReadMinSoftPosLimit(Axis := _stAxis.Axis,
                        Enable := TRUE,
                        ReadMode := READMODE_CYCLIC,
                        ParameterNumber := E_AxisParameters.SWLimitBackward,
                        Value => _stAxis.stConfig.fMinSoftPosLimit);
fbReadMaxSoftPosLimit(Axis := _stAxis.Axis,
                        Enable := TRUE,
                        ReadMode := READMODE_CYCLIC,
                        ParameterNumber := E_AxisParameters.SWLimitForward,
                        Value => _stAxis.stConfig.fMaxSoftPosLimit);

//Position Lag Monitoring
fbReadEnPositionLagMonitoring(Axis := _stAxis.Axis,
                        Enable := TRUE,
                        ReadMode := READMODE_CYCLIC,
                        ParameterNumber := E_AxisParameters.EnablePositionLagMonitoring);
_stAxis.stConfig.bEnPositionLagMonitoring := LREAL_TO_BOOL(fbReadEnPositionLagMonitoring.Value);

fbReadAxisMaxPosLagValue(Axis := _stAxis.Axis,
                        Enable := TRUE,
                        ReadMode := READMODE_CYCLIC,
                        ParameterNumber := E_AxisParameters.MaxPositionLag,
                        Value => _stAxis.stConfig.fMaxPosLagValue);

// Target Position Monitoring
fbReadEnTargetPositionMonitoring(Axis := _stAxis.Axis,
                        Enable := TRUE,
                        ReadMode := READMODE_CYCLIC,
                        ParameterNumber := E_AxisParameters.SWLimitBackward);
_stAxis.stConfig.bEnTargetPositionMonitoring := LREAL_TO_BOOL(fbReadEnTargetPositionMonitoring.Value);

fbReadTargetPositionWindow(Axis := _stAxis.Axis,
                        Enable := TRUE,
                        ReadMode := READMODE_CYCLIC,
                        ParameterNumber := E_AxisParameters.AxisTargetPositionWindow,
                        Value => _stAxis.stConfig.fTargetPositionWindow);

//All variables are valid
_stAxis.stConfig.bReadMcParametersValid := FALSE;
_stAxis.stConfig.bReadMcParametersValid := fbReadAxisVeloManSlow.Valid AND
    fbReadAxisVeloManFast.Valid AND
    fbReadHomingVelToCam.Valid AND
    fbReadHomingVelFromCam.Valid AND
    fbReadAxisVeloMax.Valid AND
    fbReadAxisAcc.Valid AND
    fbReadAxisDec.Valid AND
    fbReadEnMinSoftPosLimit.Valid AND
    fbReadEnMaxSoftPosLimit.Valid AND
    fbReadMinSoftPosLimit.Valid AND
    fbReadMaxSoftPosLimit.Valid AND
    fbReadEnPositionLagMonitoring.Valid AND
    fbReadAxisMaxPosLagValue.Valid AND
    fbReadEnTargetPositionMonitoring.Valid AND
    fbReadTargetPositionWindow.Valid;

//One of the variables has a read error
_stAxis.stConfig.bReadMcParametersError := fbReadAxisVeloManSlow.Error OR
    fbReadAxisVeloManFast.Error OR
    fbReadHomingVelToCam.Error OR
    fbReadHomingVelFromCam.Error OR
    fbReadAxisVeloMax.Error OR
    fbReadAxisAcc.Error OR
    fbReadAxisDec.Error OR
    fbReadEnMinSoftPosLimit.Error OR
    fbReadEnMaxSoftPosLimit.Error OR
    fbReadMinSoftPosLimit.Error OR
    fbReadMaxSoftPosLimit.Error OR
    fbReadEnPositionLagMonitoring.Error OR
    fbReadAxisMaxPosLagValue.Error OR
    fbReadEnTargetPositionMonitoring.Error OR
    fbReadTargetPositionWindow.Error;
END_METHOD

METHOD mParameters_ReadParameter : ST_McStatus

IF _stAxis.stControl.eCommand = E_MotionFunctions.eReadParameter THEN
    fbReadParameter.Enable := _stAxis.stControl.bExecute;
END_IF

fbReadParameter.ReadMode := E_READMODE.READMODE_ONCE;
fbReadParameter.ParameterNumber := _stAxis.stConfig.eAxisParameters;

fbReadParameter(Axis := _stAxis.Axis);
fbReadParameter.Enable := FALSE;

_stAxis.stconfig.fReadAxisParameter := fbReadParameter.Value;
mParameters_ReadParameter.Busy := fbReadParameter.Busy;
mParameters_ReadParameter.Done := fbReadParameter.Valid;
mParameters_ReadParameter.Error := fbReadParameter.Error;
mParameters_ReadParameter.ErrorID := fbReadParameter.ErrorID;

IF fbReadParameter.Error THEN
    _stAxis.stError.fbReadParameterErrorId := fbReadParameter.ErrorID;
END_IF
END_METHOD

METHOD mParameters_WriteParameter : ST_McStatus

IF _stAxis.stControl.eCommand = E_MotionFunctions.eWriteParameter THEN
    fbWriteParameter.Execute := _stAxis.stControl.bExecute;
END_IF

fbWriteParameter.ParameterNumber := _stAxis.stConfig.eAxisParameters;
fbWriteParameter.Value := _stAxis.stConfig.fWriteAxisParameter;

fbWriteParameter(Axis := _stAxis.Axis);
fbWriteParameter.Execute := FALSE;

mParameters_WriteParameter.Busy := fbWriteParameter.Busy;
mParameters_WriteParameter.Done := fbWriteParameter.Done;
mParameters_WriteParameter.Error := fbWriteParameter.Error;
mParameters_WriteParameter.ErrorID := fbWriteParameter.ErrorID;

IF fbWriteParameter.Error THEN
    _stAxis.stError.fbWriteParameterErrorId := fbWriteParameter.ErrorID;
END_IF
END_METHOD

METHOD mStatus_AxisStatus : BOOL

_stAxis.Axis.ReadStatus();
IF _stAxis.Axis.Status.OpMode.Modulo THEN
    _stAxis.stStatus.fActPosition := _stAxis.Axis.NcToPlc.ModuloActPos;
ELSE
    _stAxis.stStatus.fActPosition := _stAxis.Axis.NcToPlc.ActPos;
END_IF

_stAxis.stStatus.bHomed := _stAxis.Axis.Status.Homed;
_stAxis.stStatus.bMoving := _stAxis.Axis.Status.Moving;
_stAxis.stStatus.fActVelocity := _stAxis.Axis.NcToPlc.ActVelo;
_stAxis.stStatus.bMovingForward := _stAxis.Axis.Status.PositiveDirection;
_stAxis.stStatus.bMovingBackward := _stAxis.Axis.Status.NegativeDirection;
_stAxis.stStatus.bInTargetPosition := _stAxis.Axis.Status.InTargetPosition;
//_stAxis.stStatus.bEnabled := _stAxis.Axis.Status.Operational;
_stAxis.stStatus.bEnabled := NOT(_stAxis.Axis.Status.Disabled);	//This is crap but I don't know a better way

_stAxis.stStatus.SPGEnabled := _stAxis.Axis.Status.ExtSetPointGenEnabled;
END_METHOD

METHOD mStatus_Busy : BOOL
VAR
    i: UINT;
    tmpBusy: BOOL;
END_VAR

FOR i := 5 TO 10 DO
    tmpBusy := astMcStatus[i]^.Busy OR tmpBusy;
END_FOR
mStatus_Busy := tmpBusy;
END_METHOD

METHOD mStatus_CommandAborted : BOOL
VAR
    i: UINT;
    tmpCmdAborted: BOOL;
END_VAR

FOR i := 5 TO 9 DO
    tmpCmdAborted := astMcStatus[i]^.CommandAborted OR tmpCmdAborted;
END_FOR

fbCommandAbortedRTrig(CLK := tmpCmdAborted);
IF fbCommandAbortedRTrig.Q THEN
    _stAxis.stStatus.bCommandAborted := TRUE;
END_IF
END_METHOD

METHOD mStatus_Done : BOOL
VAR
    i: UINT;
    tmpDone: BOOL;
END_VAR

FOR i := 5 TO 10 DO
    tmpDone := astMcStatus[i]^.Done OR tmpDone;
END_FOR
//fbDoneRTrig(CLK:= mStatus_Done());
fbDoneRTrig(CLK := tmpDone);
IF fbDoneRTrig.Q THEN
    _stAxis.stStatus.bDone := TRUE;
END_IF
END_METHOD

METHOD mStatus_Error : BOOL
VAR
    i: UINT;
    tmpError: BOOL;
END_VAR

FOR i := 1 TO nMCSTATUS_ARRAY_SIZE DO
    tmpError := astMcStatus[i]^.Error OR tmpError;
END_FOR

fbErrorRTrig(CLK := tmpError);

//Check if NC is in error state and propogate
IF _stAxis.Axis.Status.ErrorStop OR _stAxis.Axis.Status.Error THEN
    _stAxis.stStatus.bError := _stAxis.Axis.Status.ErrorStop OR _stAxis.Axis.Status.Error;
    _stAxis.stStatus.nErrorID := _stAxis.Axis.Status.ErrorID;//NC Error ID
END_IF


IF fbErrorRTrig.Q THEN
        //For each mcStatus
        FOR i := 1 TO nMCSTATUS_ARRAY_SIZE DO
            //If there's an error present propagate
            IF astMcStatus[i]^.ErrorID <> 0 THEN
				_stAxis.stStatus.bMcError := TRUE;
                _stAxis.stStatus.nMcErrorID := astMcStatus[i]^.ErrorID;
            END_IF
        END_FOR
END_IF
END_METHOD

METHOD mStatus_InVelocity : BOOL
VAR
    i: UINT;
    tmpInVelocity: BOOL;
END_VAR
FOR i := 1 TO nMCSTATUS_ARRAY_SIZE DO
    tmpInVelocity := astMcStatus[i]^.InVelocity OR tmpInVelocity;
END_FOR
//fbInVelocityRTrig(CLK:= mStatus_InVelocity());
fbInVelocityRTrig(CLK := tmpInVelocity);
IF fbInVelocityRTrig.Q THEN
    _stAxis.stStatus.bInVelocity := TRUE;
END_IF

fbInVelocityFTrig(CLK := _stAxis.Axis.Status.ContinuousMotion);
IF fbInVelocityFTrig.Q THEN
    _stAxis.stStatus.bInVelocity := FALSE;
END_IF
END_METHOD

METHOD mStatus_NewCommand : BOOL
VAR
    i: UINT;
END_VAR

fbExecuteRTrig(CLK := _stAxis.stControl.bExecute);
IF fbExecuteRTrig.Q THEN
    _stAxis.stStatus.bDone := FALSE;
    _stAxis.stStatus.bCommandAborted := FALSE;

    //On a new motion command, clear the errorID
    CASE _stAxis.stControl.eCommand OF
            E_MotionFunctions.eMoveAbsolute,
            E_MotionFunctions.eMoveRelative,
            E_MotionFunctions.eMoveVelocity,
            E_MotionFunctions.eMoveModulo,
			E_MotionFunctions.eSetPosition,
            E_MotionFunctions.eHome :
                _stAxis.stStatus.nErrorID := 0;
            E_MotionFunctions.eWriteParameter,
            E_MotionFunctions.eReadParameter :
            // Nothing
    END_CASE
END_IF
END_METHOD

METHOD Run : BOOL
mStatus_AxisStatus();
mParameters_ReadNc();
mParameters_Init();
stMcStatusReadParameter := mParameters_ReadParameter();
stMcStatusWriteParameter := mParameters_WriteParameter();

mControl_LimitHitTimer();
mControl_LimitLinking();
stMcStatusPower := mControl_Power();
mControl_AutoEnableDisable();

mControl_EnableSPG();
mControl_DisableSPG();
mControl_FeedSPG();

stMcStatusHalt := mMove_Halt();
stMcStatusStop := mMove_Stop();
stMcStatusReset := mControl_Reset();
stMcStatusSetPosition := mMove_SetPosition();

stMcStatusMoveAbsolute := mMove_MoveAbsolute();
stMcStatusMoveRelative := mMove_MoveRelative();
stMcStatusMoveModulo := mMove_MoveModulo();
stMcStatusMoveVelocity := mMove_MoveVelocity();

stMcStatusHome := mControl_Home();

mStatus_NewCommand();
mStatus_Done();
mStatus_Error();
mStatus_InVelocity();
mStatus_CommandAborted();
_stAxis.stStatus.bBusy := mStatus_Busy();


EndOfCycle();
END_METHOD

PROPERTY stAxis : REFERENCE TO ST_AxisStruct
GET
stAxis REF= _stAxis;
END_GET
SET
_stAxis REF= stAxis;
END_SET
END_PROPERTY

END_FUNCTION_BLOCK

// ---- tc_mca_std_lib/VISUs/MainVisu.TcVIS
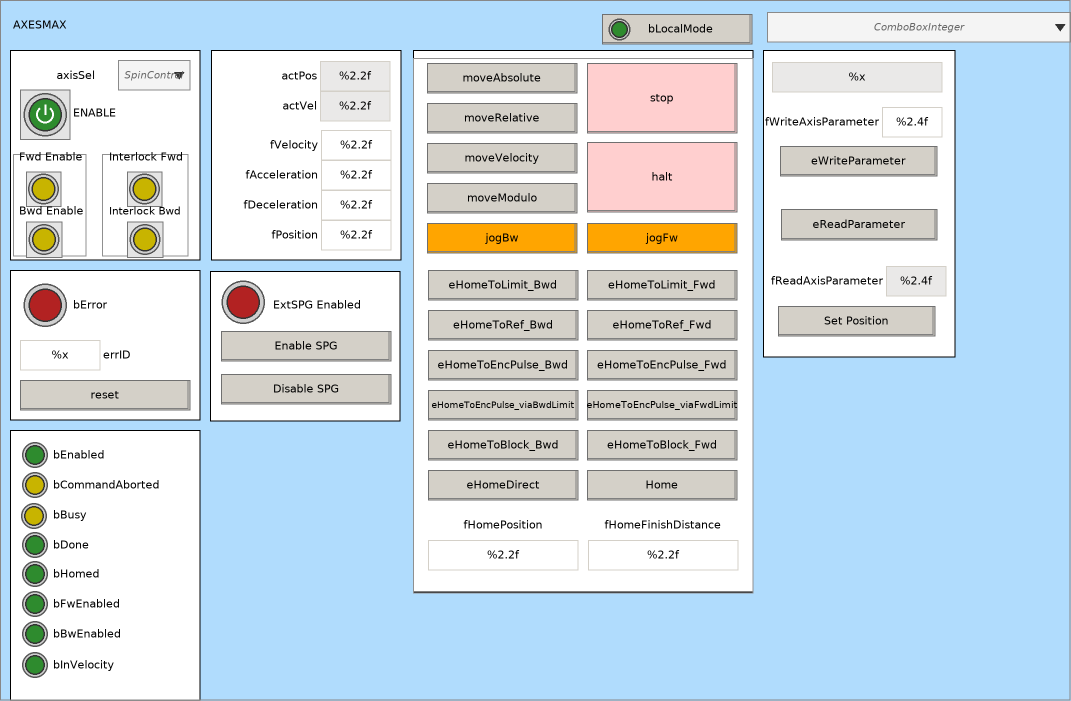
VISUALIZATION MainVisu  // 1071x701
    Rectangle (210,271 190x150)
    Rectangle (413,50 340x542)
    GroupBox (413,50 340x543)
        Button (174,92 150x70), "halt", pressed state: GVL.astAxes[Main.hmiAxisSelection].stControl.bHalt, text list: "languageSupport", text index: "halt"
            toggle GVL.astAxes[Main.hmiAxisSelection].stControl.bHalt
        Button (174,420 150x30), "Home", text list: 'languageSupport', text index: "Home"
            OnMouseClick: execute { GVL.astAxes[Main.hmiAxisSelection].stControl.eCommand:=E_MotionFunctions.eHome; GVL.astAxes[Main.hmiAxisSelection].stControl.bExecute:=TRUE; }
        Button (15,380 150x30), "eHomeToBlock_Bwd", text list: 'languageSupport', text index: "eHomeToBlock_Bwd"
            OnMouseClick: execute {
                GVL.astAxes[Main.hmiAxisSelection].stControl.eCommand:=E_MotionFunctions.eHome;
                GVL.astAxes[Main.hmiAxisSelection].stHomingConfig.eHomeSeq:=E_HomingRoutines.eHomeToBlock_Bwd;
                GVL.astAxes[Main.hmiAxisSelection].stControl.bExecute:=TRUE;
            }
    GroupBox (10,50 190x210)
        Rectangle (0,0 190x210)
        GroupBox (3,96 73x110)
        GroupBox (92,96 86x110)
        Textfield (60,50 92x26), "ENABLE", text list: 'languageSupport', text index: "enable"
        PushSwitchLed (16,118 35x42), variable: GVL.astAxes[MAIN.hmiAxisSelection].stInputs.bLimitFwd, behaviour: TOGGLE, style: Switch-PushSwitchLed-Yellow
        PushSwitchLed (16,170 36x39), variable: GVL.astAxes[MAIN.hmiAxisSelection].stInputs.bLimitBwd, behaviour: TOGGLE, style: Switch-PushSwitchLed-Yellow
        SpinControl (108,10 72x30), variable: MAIN.hmiAxisSelection
            p651134158: GVL_APP.nAXIS_NUM
        Textfield (23,13 86x25), "axisSel", text variable: GVL_APP.nAXIS_NUM, text list: "languageSupport", text index: "axisSel"
        PowerSwitch (10,38 50x53), variable: GVL.astAxes[MAIN.hmiAxisSelection].stControl.bEnable, behaviour: TOGGLE, style: Switch-PowerSwitch-Green
        PushSwitchLed (117,118 35x42), variable: GVL.astAxes[MAIN.hmiAxisSelection].stControl.bInterlockFwd, behaviour: TOGGLE, style: Switch-PushSwitchLed-Yellow
        PushSwitchLed (117,170 36x39), variable: GVL.astAxes[MAIN.hmiAxisSelection].stControl.bInterlockBwd, behaviour: TOGGLE, style: Switch-PushSwitchLed-Yellow
        Textfield (6,94 76x26), "Fwd Enable", text list: 'languageSupport', text index: "enFW"
        Textfield (6,148 76x26), "Bwd Enable", text list: 'languageSupport', text index: "enBW"
        Textfield (96,94 76x26), "Interlock Fwd", text list: 'languageSupport', text index: "bAxisInterlockFwd"
        Textfield (96,148 76x26), "Interlock Bwd", text list: 'languageSupport', text index: "bAxisInterlockBwd"
    Textfield (10,10 231x30), "AXESMAX", text variable: GVL_APP.nAXIS_NUM, text list: "languageSupport", text index: "axesAvailable"
    Button (427,63 150x30), "moveAbsolute", text list: "languageSupport", text index: "moveAbsolute"
        OnMouseClick: execute { GVL.astAxes[MAIN.hmiAxisSelection].stControl.eCommand:=E_MotionFunctions.eMoveAbsolute; GVL.astAxes[MAIN.hmiAxisSelection].stControl.bExecute:=TRUE; }
    Button (427,143 150x30), "moveVelocity", text list: "languageSupport", text index: "moveVelocity"
        OnMouseClick: execute { GVL.astAxes[Main.hmiAxisSelection].stControl.eCommand:=E_MotionFunctions.eMoveVelocity; GVL.astAxes[Main.hmiAxisSelection].stControl.bExecute:=TRUE; }
    Button (427,103 150x30), "moveRelative", text list: "languageSupport", text index: "moveRelative"
        OnMouseClick: execute { GVL.astAxes[Main.hmiAxisSelection].stControl.eCommand:=E_MotionFunctions.eMoveRelative; GVL.astAxes[Main.hmiAxisSelection].stControl.bExecute:=TRUE; }
    Button (427,183 150x30), "moveModulo", text list: "languageSupport", text index: "moveModulo"
        OnMouseClick: execute { GVL.astAxes[Main.hmiAxisSelection].stControl.eCommand:=E_MotionFunctions.eMoveModulo; GVL.astAxes[Main.hmiAxisSelection].stControl.bExecute:=TRUE; }
    Button (587,63 150x70), "stop", pressed state: GVL.astAxes[Main.hmiAxisSelection].stControl.bStop, text list: "languageSupport", text index: "stop"
        toggle GVL.astAxes[Main.hmiAxisSelection].stControl.bStop
    Button (427,223 150x30), "jogBw", text list: "languageSupport", text index: "jogBw"
        OnMouseDown: execute {
            GVL.astAxes[Main.hmiAxisSelection].stControl.eCommand:=E_MotionFunctions.eMoveVelocity;
            GVL.astAxes[Main.hmiAxisSelection].stControl.fVelocity:=-ABS(GVL.astAxes[Main.hmiAxisSelection].stControl.fJogVelocity)
            GVL.astAxes[Main.hmiAxisSelection].stControl.bExecute:= TRUE;
        }
        OnMouseClick: execute {  }
        OnMouseUp: execute { GVL.astAxes[Main.hmiAxisSelection].stControl.bHalt:= TRUE; }
    Button (587,223 150x30), "jogFw", text list: "languageSupport", text index: "jogFw"
        OnMouseDown: execute {
            GVL.astAxes[Main.hmiAxisSelection].stControl.eCommand:=E_MotionFunctions.eMoveVelocity;
            GVL.astAxes[Main.hmiAxisSelection].stControl.fVelocity:=ABS(GVL.astAxes[Main.hmiAxisSelection].stControl.fJogVelocity)
            GVL.astAxes[Main.hmiAxisSelection].stControl.bExecute:= TRUE;
        }
        OnMouseClick: execute {  }
        OnMouseUp: execute { GVL.astAxes[Main.hmiAxisSelection].stControl.bHalt:= TRUE; }
    GroupBox (10,270 190x150)
        Rectangle (0,0 190x150)
        Textfield (90,70 90x30), "errID", text list: "languageSupport", text index: "errID"
        Textfield (10,70 80x30), "%x", text variable: GVL.astAxes[MAIN.hmiAxisSelection].stStatus.nErrorID
        Lamp1 (10,10 50x50), variable: GVL.astAxes[MAIN.hmiAxisSelection].stStatus.bError, style: Lamp-Lamp1-Red
        Textfield (60,20 120x30), "bError", text list: "languageSupport", text index: "bError"
        Button (10,110 170x30), "reset", pressed state: GVL.astAxes[Main.hmiAxisSelection].stControl.bReset, text list: "languageSupport", text index: "reset"
            OnMouseClick: toggle GVL.astAxes[Main.hmiAxisSelection].stControl.bReset
    GroupBox (10,430 190x271)
        Rectangle (0,0 190x270)
        Lamp1 (10,10 30x30), variable: GVL.astAxes[MAIN.hmiAxisSelection].stStatus.bEnabled, style: Lamp-Lamp1-Green
        Textfield (40,10 140x30), "bEnabled", text list: "languageSupport", text index: "bEnabled"
        Lamp1 (10,40 30x30), variable: GVL.astAxes[MAIN.hmiAxisSelection].stStatus.bCommandAborted, style: Lamp-Lamp1-Yellow
        Textfield (40,40 140x30), "bCommandAborted", text list: "languageSupport", text index: "bWarning"
        Textfield (40,70 140x30), "bBusy", text list: "languageSupport", text index: "bBusy"
        Lamp1 (10,100 30x30), variable: GVL.astAxes[MAIN.hmiAxisSelection].stStatus.bDone, style: Lamp-Lamp1-Green
        Textfield (40,100 140x30), "bDone", text list: 'languageSupport', text index: "bDone"
        Lamp1 (10,129 30x30), variable: GVL.astAxes[MAIN.hmiAxisSelection].stStatus.bHomed, style: Lamp-Lamp1-Green
        Textfield (40,129 140x30), "bHomed", text list: "languageSupport", text index: "bHomed"
        Lamp1 (10,159 30x30), variable: GVL.astAxes[MAIN.hmiAxisSelection].stStatus.bFwEnabled AND NOT GVL.astAxes[MAIN.hmiAxisSelection].stStatus.bInterlockedFwd, style: Lamp-Lamp1-Green
        Lamp1 (10,189 30x30), variable: GVL.astAxes[MAIN.hmiAxisSelection].stStatus.bBwEnabled AND NOT GVL.astAxes[MAIN.hmiAxisSelection].stStatus.bInterlockedBwd, style: Lamp-Lamp1-Green
        Textfield (40,159 140x30), "bFwEnabled", text list: "languageSupport", text index: "bFwEnabled"
        Textfield (40,189 140x30), "bBwEnabled", text list: "languageSupport", text index: "bBwEnabled"
        Lamp1 (9,71 30x30), variable: GVL.astAxes[MAIN.hmiAxisSelection].stStatus.bBusy, style: Lamp-Lamp1-Yellow
        Lamp1 (10,220 30x30), variable: GVL.astAxes[MAIN.hmiAxisSelection].stStatus.bInVelocity, style: Lamp-Lamp1-Green
    GroupBox (211,50 190x210)
        Rectangle (0,0 190x210)
        Textfield (10,80 100x30), "fVelocity", text list: "languageSupport", text index: "fVelocity"
        Textfield (110,80 70x30), "%2.2f", text variable: GVL.astAxes[MAIN.hmiAxisSelection].stControl.fVelocity
            OnMouseClick: write the text variable via Default
        Textfield (10,110 100x30), "fAcceleration", text list: "languageSupport", text index: "fAcceleration"
        Textfield (110,110 70x30), "%2.2f", text variable: GVL.astAxes[MAIN.hmiAxisSelection].stControl.fAcceleration
            OnMouseClick: write the text variable via Default
        Textfield (10,140 100x30), "fDeceleration", text list: "languageSupport", text index: "fDeceleration"
        Textfield (110,140 70x30), "%2.2f", text variable: GVL.astAxes[MAIN.hmiAxisSelection].stControl.fDeceleration
            OnMouseClick: write the text variable via Default
        Textfield (10,170 100x30), "fPosition", text list: "languageSupport", text index: "fPosition"
        Textfield (110,170 70x30), "%2.2f", text variable: GVL.astAxes[MAIN.hmiAxisSelection].stControl.fPosition
            OnMouseClick: write the text variable via Default
        Textfield (109,11 70x30), "%2.2f", text variable: GVL.astAxes[MAIN.hmiAxisSelection].stStatus.fActPosition
        Textfield (9,11 100x30), "actPos", text list: "languageSupport", text index: "actposition"
        Textfield (9,41 100x30), "actVel", text list: "languageSupport", text index: "actVelocity"
        Textfield (109,41 70x30), "%2.2f", text variable: GVL.astAxes[MAIN.hmiAxisSelection].stStatus.fActVelocity
    Button (428,310 150x30), "eHomeToRef_Bwd", text list: 'languageSupport', text index: "eHomeToRef_Bwd"
        OnMouseClick: execute {
            GVL.astAxes[Main.hmiAxisSelection].stControl.eCommand:=E_MotionFunctions.eHome;
            GVL.astAxes[Main.hmiAxisSelection].stHomingConfig.eHomeSeq:=E_HomingRoutines.eHomeToRef_Bwd;
            GVL.astAxes[Main.hmiAxisSelection].stControl.bExecute:=TRUE;
        }
    Button (587,310 150x30), "eHomeToRef_Fwd", text list: "languageSupport", text index: "eHomeToRef_Fwd"
        OnMouseClick: execute {
            GVL.astAxes[Main.hmiAxisSelection].stControl.eCommand:=E_MotionFunctions.eHome;
            GVL.astAxes[Main.hmiAxisSelection].stHomingConfig.eHomeSeq:=E_HomingRoutines.eHomeToRef_Fwd;
            GVL.astAxes[Main.hmiAxisSelection].stControl.bExecute:=TRUE;
        }
    Button (428,350 150x30), "eHomeToEncPulse_Bwd", text list: 'languageSupport', text index: "eHomeToEncPulse_Bwd"
        OnMouseClick: execute {
            GVL.astAxes[Main.hmiAxisSelection].stControl.eCommand:=E_MotionFunctions.eHome;
            GVL.astAxes[Main.hmiAxisSelection].stHomingConfig.eHomeSeq:=E_HomingRoutines.eHomeToEncPulse_Bwd;
            GVL.astAxes[Main.hmiAxisSelection].stControl.bExecute:=TRUE;
        }
    Button (587,350 150x30), "eHomeToEncPulse_Fwd", text list: "languageSupport", text index: "eHomeToEncPulse_Fwd"
        OnMouseClick: execute {
            GVL.astAxes[Main.hmiAxisSelection].stControl.eCommand:=E_MotionFunctions.eHome;
            GVL.astAxes[Main.hmiAxisSelection].stHomingConfig.eHomeSeq:=E_HomingRoutines.eHomeToEncPulse_Fwd;
            GVL.astAxes[Main.hmiAxisSelection].stControl.bExecute:=TRUE;
        }
    Button (428,470 150x30), "eHomeDirect", text list: 'languageSupport', text index: "eHomeDirect"
        OnMouseClick: execute {
            GVL.astAxes[Main.hmiAxisSelection].stControl.eCommand:=E_MotionFunctions.eHome;
            GVL.astAxes[Main.hmiAxisSelection].stHomingConfig.eHomeSeq:=E_HomingRoutines.eHomeDirect;
            GVL.astAxes[Main.hmiAxisSelection].stControl.bExecute:=TRUE;
        }
    Button (428,270 150x30), "eHomeToLimit_Bwd", text list: 'languageSupport', text index: "eHomeToLimit_Bwd"
        OnMouseClick: execute {
            GVL.astAxes[Main.hmiAxisSelection].stControl.eCommand:=E_MotionFunctions.eHome;
            GVL.astAxes[Main.hmiAxisSelection].stHomingConfig.eHomeSeq:=E_HomingRoutines.eHomeToLimit_Bwd;
            GVL.astAxes[Main.hmiAxisSelection].stControl.bExecute:=TRUE;
        }
    Button (587,270 150x30), "eHomeToLimit_Fwd", text list: "languageSupport", text index: "eHomeToLimit_Fwd"
        OnMouseClick: execute {
            GVL.astAxes[Main.hmiAxisSelection].stControl.eCommand:=E_MotionFunctions.eHome;
            GVL.astAxes[Main.hmiAxisSelection].stHomingConfig.eHomeSeq:=E_HomingRoutines.eHomeToLimit_Fwd;
            GVL.astAxes[Main.hmiAxisSelection].stControl.bExecute:=TRUE;
        }
    Textfield (428,540 150x30), "%2.2f", text variable: GVL.astAxes[MAIN.hmiAxisSelection].stHomingConfig.fHomePosition
        OnMouseClick: write GVL.astAxes[MAIN.hmiAxisSelection].stHomingConfig.fHomePosition via Default
    Button (428,390 150x30), "eHomeToEncPulse_viaBwdLimit", text list: 'languageSupport', text index: "eHomeToEncPulse_viaBwdLimit"
        OnMouseClick: execute {
            GVL.astAxes[Main.hmiAxisSelection].stControl.eCommand:=E_MotionFunctions.eHome;
            GVL.astAxes[Main.hmiAxisSelection].stHomingConfig.eHomeSeq:=E_HomingRoutines.eHomeToEncPulse_viaBwdLimit;
            GVL.astAxes[Main.hmiAxisSelection].stControl.bExecute:=TRUE;
        }
    Button (587,390 150x30), "eHomeToEncPulse_viaFwdLimit", text list: "languageSupport", text index: "eHomeToEncPulse_viaFwdLimit"
        OnMouseClick: execute {
            GVL.astAxes[Main.hmiAxisSelection].stControl.eCommand:=E_MotionFunctions.eHome;
            GVL.astAxes[Main.hmiAxisSelection].stHomingConfig.eHomeSeq:=E_HomingRoutines.eHomeToEncPulse_viaFwdLimit;
            GVL.astAxes[Main.hmiAxisSelection].stControl.bExecute:=TRUE;
        }
    Textfield (588,540 150x30), "%2.2f", text variable: GVL.astAxes[MAIN.hmiAxisSelection].stHomingConfig.fHomeFinishDistance, text list: ''
        OnMouseClick: write GVL.astAxes[MAIN.hmiAxisSelection].stHomingConfig.fHomeFinishDistance via Default
    Textfield (428,510 150x30), "fHomePosition", text list: "languageSupport", text index: "fHomePosition"
    Textfield (588,510 150x30), "fHomeFinishDistance", text list: "languageSupport", text index: "fHomeFinishDistance"
    Group (602,14 150x30)
        Button (0,0 150x30), "bLocalMode", text list: 'languageSupport', text index: bLocalMode
            OnMouseClick: toggle bLocalMode
        Lamp1 (5,3 25x25), variable: bLocalMode, style: Lamp-Lamp1-Green
    Rectangle (763,50 192x307)
    Button (780,146 157x30), "eWriteParameter", text list: "languageSupport", text index: "eWriteParameter"
        OnMouseClick: execute { GVL.astAxes[MAIN.hmiAxisSelection].stControl.eCommand:=E_MotionFunctions.eWriteParameter; GVL.astAxes[MAIN.hmiAxisSelection].stControl.bExecute:=TRUE; }
    Textfield (772,62 170x30), "%x", text variable: astAxes[MAIN.hmiAxisSelection].stConfig.eAxisParameters
        OnMouseClick: write GVL.astAxes[MAIN.hmiAxisSelection].stConfig.eAxisParameters via Default
    Textfield (762,107 120x30), "fWriteAxisParameter", text list: "languageSupport", text index: "fWriteAxisParameter"
    Textfield (882,107 60x30), "%2.4f", text variable: astAxes[MAIN.hmiAxisSelection].stConfig.fWriteAxisParameter
        OnMouseClick: write GVL.astAxes[MAIN.hmiAxisSelection].stConfig.fWriteAxisParameter via Default
    Textfield (886,266 60x30), "%2.4f", text variable: astAxes[MAIN.hmiAxisSelection].stConfig.fReadAxisParameter
        OnMouseClick: write GVL.astAxes[MAIN.hmiAxisSelection].stConfig.fReadAxisParameter via Default
    Textfield (766,266 120x30), "fReadAxisParameter", text list: "languageSupport", text index: "fReadAxisParameter"
    Button (781,209 156x31), "eReadParameter", text list: 'languageSupport', text index: "eReadParameter"
        OnMouseClick: execute { GVL.astAxes[MAIN.hmiAxisSelection].stControl.eCommand:=E_MotionFunctions.eReadParameter; GVL.astAxes[MAIN.hmiAxisSelection].stControl.bExecute:=TRUE; }
    ComboBoxInteger (767,12 304x30), variable: GVL.astAxes[MAIN.hmiAxisSelection].stConfig.eAxisParameters, text list: 'ParameterTextList'
    Textfield (50,650 140x30), "bInVelocity", text list: 'languageSupport', text index: "bInVelocity"
    Button (587,430 150x30), "eHomeToBlock_Fwd", text list: "languageSupport", text index: "eHomeToBlock_Fwd"
        OnMouseClick: execute {
            GVL.astAxes[Main.hmiAxisSelection].stControl.eCommand:=E_MotionFunctions.eHome;
            GVL.astAxes[Main.hmiAxisSelection].stHomingConfig.eHomeSeq:=E_HomingRoutines.eHomeToBlock_Fwd;
            GVL.astAxes[Main.hmiAxisSelection].stControl.bExecute:=TRUE;
        }
    Textfield (270,290 120x30), "ExtSPG Enabled", text list: "languageSupport", text index: "bError"
    Lamp1 (218,277 50x50), variable: GVL.astAxes[MAIN.hmiAxisSelection].stStatus.SPGEnabled, style: Lamp-Lamp1-Red
    Button (221,331 170x30), "Enable SPG", pressed state: GVL.astAxes[Main.hmiAxisSelection].stControl.bReset, text list: "languageSupport", text index: "reset"
        OnMouseClick: toggle GVL.astAxes[Main.hmiAxisSelection].stSpg.EnableSPG
    Button (221,374 170x30), "Disable SPG", pressed state: GVL.astAxes[Main.hmiAxisSelection].stControl.bReset, text list: "languageSupport", text index: "reset"
        OnMouseClick: toggle GVL.astAxes[Main.hmiAxisSelection].stSpg.DisableSPG
    Button (778,306 157x30), "Set Position", text list: "languageSupport", text index: "eWriteParameter"
        OnMouseClick: execute { GVL.astAxes[MAIN.hmiAxisSelection].stControl.eCommand:=E_MotionFunctions.eSetPosition; GVL.astAxes[MAIN.hmiAxisSelection].stControl.bExecute:=TRUE; }
END_VISUALIZATION

// ---- tc_mca_std_lib/VISUs/PneumaticsVisu.TcVIS
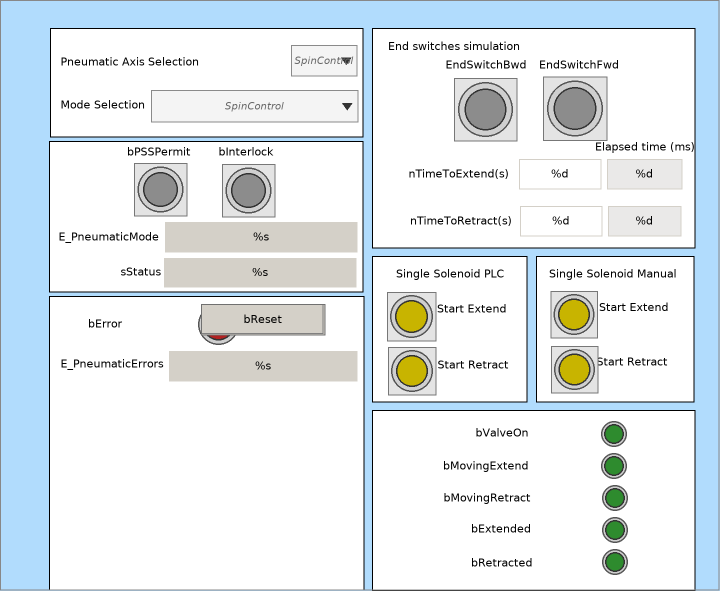
VISUALIZATION PneumaticsVisu  // 720x591
    Rectangle (50,28 313x109)
    Label (55,47 150x30), "Pneumatic Axis Selection"
    Rectangle (372,28 323x220)
    Label (379,30 150x33), "End switches simulation"
    Label (411,50 150x30), "EndSwitchBwd"
    SpinControl (291,45 66x31), variable: MAIN.hmiPneumaticAxisSelection
        p651134158: GVL_APP.nPNEUMATIC_AXIS_NUM
    Label (504,50 150x30), "EndSwitchFwd"
    Rectangle (49,296 315x294)
    Textfield (519,159 82x30), "%d", text variable: MAIN.afbPneumaticAxes[MAIN.hmiPneumaticAxisSelection].stPneumaticAxisStruct.stPneumaticAxisConfig.nTimeToExtend
        OnMouseClick: write MAIN.afbPneumaticAxes[MAIN.hmiPneumaticAxisSelection].stPneumaticAxisStruct.stPneumaticAxisConfig.nTimeToExtend via Default
    Label (384,159 150x30), "nTimeToExtend(s)"
    Label (386,206 150x30), "nTimeToRetract(s)"
    Label (28,90 150x30), "Mode Selection"
    Rectangle (49,141 314x151)
    Label (30,309 150x30), "bError"
    Lamp1 (126,301 185x47), variable: MAIN.afbPneumaticAxes[MAIN.hmiPneumaticAxisSelection].stPneumaticAxisStruct.stPneumaticAxisStatus.bError, style: Lamp-Lamp1-Red
    Label (37,349 150x30), "E_PneumaticErrors"
    Textfield (169,351 188x30), "%s", text variable: MAIN.afbPneumaticAxes[MAIN.hmiPneumaticAxisSelection].stPneumaticAxisStruct.ePneumaticAxisErrors, text list: 'languageSupport'
    Rectangle (372,256 155x146)
    Rectangle (536,256 158x146)
    Rectangle (372,410 323x181)
    Label (538,259 150x30), "Single Solenoid Manual"
    PushSwitchLed (549,291 50x47), variable: MAIN.afbPneumaticAxes[MAIN.hmiPneumaticAxisSelection].stPneumaticAxisStruct.stPneumaticAxisInputs.bOpenManual, behaviour: TOGGLE, style: Switch-PushSwitchLed-Yellow
    Label (592,293 84x29), "Start Extend"
    Label (557,347 150x30), "Start Retract"
    Label (375,259 150x30), "Single Solenoid PLC"
    PushSwitchLed (387,292 49x49), variable: MAIN.afbPneumaticAxes[MAIN.hmiPneumaticAxisSelection].stPneumaticAxisStruct.stPneumaticAxisControl.bExtend, behaviour: TOGGLE, style: Switch-PushSwitchLed-Yellow
    PushSwitchLed (388,347 48x48), variable: MAIN.afbPneumaticAxes[MAIN.hmiPneumaticAxisSelection].stPneumaticAxisStruct.stPneumaticAxisControl.bRetract, behaviour: TOGGLE, style: Switch-PushSwitchLed-Yellow
    Label (427,418 150x30), "bValveOn"
    Lamp1 (539,419 150x30), variable: MAIN.afbPneumaticAxes[MAIN.hmiPneumaticAxisSelection].stPneumaticAxisStruct.stPneumaticAxisOutputs.bValveOn, style: Lamp-Lamp1-Green
    Label (411,451 150x30), "bMovingExtend"
    Lamp1 (539,451 150x30), variable: MAIN.afbPneumaticAxes[MAIN.hmiPneumaticAxisSelection].stPneumaticAxisStruct.stPneumaticAxisStatus.bExtending, style: Lamp-Lamp1-Green
    Lamp1 (540,483 150x30), variable: MAIN.afbPneumaticAxes[MAIN.hmiPneumaticAxisSelection].stPneumaticAxisStruct.stPneumaticAxisStatus.bRetracting, style: Lamp-Lamp1-Green
    Lamp1 (540,515 150x30), variable: MAIN.afbPneumaticAxes[MAIN.hmiPneumaticAxisSelection].stPneumaticAxisStruct.stPneumaticAxisStatus.bExtended, style: Lamp-Lamp1-Green
    Lamp1 (540,547 150x30), variable: MAIN.afbPneumaticAxes[MAIN.hmiPneumaticAxisSelection].stPneumaticAxisStruct.stPneumaticAxisStatus.bRetracted, style: Lamp-Lamp1-Green
    Label (412,483 150x30), "bMovingRetract"
    Label (426,514 150x30), "bExtended"
    Label (397,294 150x30), "Start Extend"
    Label (398,350 150x30), "Start Retract"
    Label (427,548 150x30), "bRetracted"
    Button (201,304 124x31), "bReset"
        toggle MAIN.afbPneumaticAxes[MAIN.hmiPneumaticAxisSelection].stPneumaticAxisStruct.stPneumaticAxisControl.bReset
    PushSwitchLed (549,346 51x47), variable: MAIN.afbPneumaticAxes[MAIN.hmiPneumaticAxisSelection].stPneumaticAxisStruct.stPneumaticAxisInputs.bCloseManual, behaviour: TOGGLE, style: Switch-PushSwitchLed-Yellow
    Label (84,137 150x30), "bPSSPermit"
    Label (34,222 150x30), "E_PneumaticMode"
    Textfield (165,222 192x30), "%s", text variable: MAIN.afbPneumaticAxes[MAIN.hmiPneumaticAxisSelection].stPneumaticAxisStruct.ePneumaticAxisMode, text list: 'languageSupport'
    Textfield (164,258 192x29), "%s", text variable: MAIN.afbPneumaticAxes[MAIN.hmiPneumaticAxisSelection].stPneumaticAxisStruct.stPneumaticAxisStatus.sStatus, text list: 'languageSupport'
    Label (66,257 150x30), "sStatus"
    Textfield (520,206 82x30), "%d", text variable: MAIN.afbPneumaticAxes[MAIN.hmiPneumaticAxisSelection].stPneumaticAxisStruct.stPneumaticAxisConfig.nTimeToRetract
        OnMouseClick: write MAIN.afbPneumaticAxes[MAIN.hmiPneumaticAxisSelection].stPneumaticAxisStruct.stPneumaticAxisConfig.nTimeToRetract via Default
    Textfield (607,159 75x30), "%d", text variable: MAIN.afbPneumaticAxes[MAIN.hmiPneumaticAxisSelection].fbTimerExtend.ET
    Textfield (608,206 73x30), "%d", text variable: MAIN.afbPneumaticAxes[MAIN.hmiPneumaticAxisSelection].fbTimerRetract.ET
    SpinControl (151,90 207x32), variable: MAIN.afbPneumaticAxes[MAIN.hmiPneumaticAxisSelection].stPneumaticAxisStruct.ePneumaticAxisMode
    Label (570,132 150x30), "Elapsed time (ms)"
    PushSwitchLed (454,77 63x65), variable: MAIN.afbPneumaticAxes[MAIN.hmiPneumaticAxisSelection].stPneumaticAxisStruct.stPneumaticAxisInputs.bEndSwitchBwd, behaviour: TOGGLE, style: Switch-PushSwitchLed-Gray
    PushSwitchLed (543,76 64x65), variable: MAIN.afbPneumaticAxes[MAIN.hmiPneumaticAxisSelection].stPneumaticAxisStruct.stPneumaticAxisInputs.bEndSwitchFwd, behaviour: TOGGLE, style: Switch-PushSwitchLed-Gray
    PushSwitchLed (134,163 53x53), variable: MAIN.afbPneumaticAxes[MAIN.hmiPneumaticAxisSelection].stPneumaticAxisStruct.stPneumaticAxisInputs.bPSSPermit, behaviour: TOGGLE, style: Switch-PushSwitchLed-Gray
    PushSwitchLed (222,164 53x53), variable: MAIN.afbPneumaticAxes[MAIN.hmiPneumaticAxisSelection].stPneumaticAxisStruct.stPneumaticAxisControl.bInterlock, behaviour: TOGGLE, style: Switch-PushSwitchLed-Gray
    Label (171,137 150x30), "bInterlock"
END_VISUALIZATION
